output.Value := FALSE;
Assert.ThatBool(
	actual := output.Changed,
	message := "The reverse transition must also be pending"
).IsTrue();
output.ProcessOutput();
Assert.ThatBool(
	actual := output.Changed,
	message := "Processing acknowledges the reverse transition"
).IsFalse();
Assert.ThatBool(
	actual := rawOutput,
	message := "rawOutput should be FALSE"
).IsFalse();
END_METHOD

//! <summary>Borrows the concrete class name. Callers must not modify it.</summary>
{attribute 'monitoring' := 'call'}
PROPERTY ClassName : REFERENCE TO STRING
GET
ClassName REF= _ClassName;
END_GET
END_PROPERTY

//! <summary>Borrows the compiler-initialized namespace name. Callers must not modify it.</summary>
{attribute 'monitoring' := 'call'}
PROPERTY NamespaceName : REFERENCE TO STRING
GET
NamespaceName REF= CurrentNamespace.Name;
END_GET
END_PROPERTY

//! <summary>Reports the concrete instance size in bytes.</summary>
{attribute 'monitoring' := 'call'}
PROPERTY SelfSize : ULINT
GET
SelfSize := XSIZEOF(THIS^);
END_GET
END_PROPERTY

END_FUNCTION_BLOCK

// ---- Tests/Devices/IO/DigitalOutputNormallyClosedTest.TcPOU
(*
SPDX-FileCopyrightText: c 2026 Oleksandr Tiutyk <trofimich@gmail.com>
SPDX-License-Identifier: MIT
License: https://opensource.org/license/mit
*)

(*!
<summary>Checks normally closed output inversion in both directions.</summary>
<description>
Uses a live case-owned automation parent and fresh local device fixtures on every run.
The scenario reads and writes ordinary simulated storage within one task cycle.
</description>
*)

{attribute 'no_assign'}
{attribute 'no_explicit_call' := 'do not call this function block directly'}
FUNCTION_BLOCK DigitalOutputNormallyClosedTest EXTENDS TOF_Testing.SingleCycleTest
VAR_STAT
	{attribute 'hide'}
	_ClassName : STRING := __POUNAME();
END_VAR
VAR
	//! <summary>Live parent borrowed by the method-local simulated device.</summary>
	_AutomationRoot : MockAutomationController(name := "DevicesIORoot");
END_VAR

(*!
<summary>Checks normally closed output inversion in both directions.</summary>
*)
METHOD PROTECTED ExecuteTest
VAR
	output : TOF_Devices_IO.DigitalOutput(name := "DO_NC", parent := _AutomationRoot);
	rawOutput : BOOL;
END_VAR
output.Initialize();
output.ContactType := TOF_Devices_IO.CONTACT_TYPE.NORMALLY_CLOSED;
output.BindToIO(rawValue := rawOutput);

output.Value := TRUE;
output.ProcessOutput();
Assert.ThatBool(
	actual := rawOutput,
	message := "rawOutput should be inverted FALSE for NC contact"
).IsFalse();

output.Value := FALSE;
output.ProcessOutput();
Assert.ThatBool(
	actual := rawOutput,
	message := "rawOutput should be inverted TRUE for NC contact"
).IsTrue();
END_METHOD

//! <summary>Borrows the concrete class name. Callers must not modify it.</summary>
{attribute 'monitoring' := 'call'}
PROPERTY ClassName : REFERENCE TO STRING
GET
ClassName REF= _ClassName;
END_GET
END_PROPERTY

//! <summary>Borrows the compiler-initialized namespace name. Callers must not modify it.</summary>
{attribute 'monitoring' := 'call'}
PROPERTY NamespaceName : REFERENCE TO STRING
GET
NamespaceName REF= CurrentNamespace.Name;
END_GET
END_PROPERTY

//! <summary>Reports the concrete instance size in bytes.</summary>
{attribute 'monitoring' := 'call'}
PROPERTY SelfSize : ULINT
GET
SelfSize := XSIZEOF(THIS^);
END_GET
END_PROPERTY

END_FUNCTION_BLOCK

// ---- Tests/Devices/IO/DirectAnalogValueConverterTest.TcPOU
(*
SPDX-FileCopyrightText: c 2026 Oleksandr Tiutyk <trofimich@gmail.com>
SPDX-License-Identifier: MIT
License: https://opensource.org/license/mit
*)

(*!
<summary>Checks direct conversion of INT16, INT32 and REAL32 in both directions.</summary>
<description>
Uses fresh method-local fixtures in a single task cycle.
</description>
*)

{attribute 'no_assign'}
{attribute 'no_explicit_call' := 'do not call this function block directly'}
FUNCTION_BLOCK DirectAnalogValueConverterTest EXTENDS TOF_Testing.SingleCycleTest
VAR_STAT
	{attribute 'hide'}
	_ClassName : STRING := __POUNAME();
END_VAR

(*!
<summary>Checks direct conversion of INT16, INT32 and REAL32 in both directions.</summary>
*)
METHOD PROTECTED ExecuteTest
VAR
	converter : TOF_Devices_IO.DirectAnalogValueConverter;
	rawResult : TOF_Devices_IO.RAW_ANALOG_VALUE;
	engineeringValue : LREAL;
END_VAR
// INT16
rawResult := converter.ConvertAnalogValueToRawValue(
	analogValue := 1234.0,
	rawValueType := TOF_Devices_IO.RAW_ANALOG_VALUE_TYPE.INT16
);
Assert.ThatInt(
	actual := rawResult.Int16,
	message := "INT16 raw value 1:1"
).ToBe(expected := 1234);

engineeringValue := converter.ConvertRawValueToAnalogValue(
	rawValue := rawResult,
	rawValueType := TOF_Devices_IO.RAW_ANALOG_VALUE_TYPE.INT16
);
Assert.ThatLongReal(
	actual := engineeringValue,
	message := "INT16 analog value 1:1"
).ToBe(expected := 1234.0, tolerance := 0.001);

// INT32
rawResult := converter.ConvertAnalogValueToRawValue(
	analogValue := 100000.0,
	rawValueType := TOF_Devices_IO.RAW_ANALOG_VALUE_TYPE.INT32
);
Assert.ThatDInt(
	actual := rawResult.Int32,
	message := "INT32 raw value 1:1"
).ToBe(expected := 100000);

engineeringValue := converter.ConvertRawValueToAnalogValue(
	rawValue := rawResult,
	rawValueType := TOF_Devices_IO.RAW_ANALOG_VALUE_TYPE.INT32
);
Assert.ThatLongReal(
	actual := engineeringValue,
	message := "INT32 analog value 1:1"
).ToBe(expected := 100000.0, tolerance := 0.001);

// REAL32 preserves both sign and fraction.
rawResult := converter.ConvertAnalogValueToRawValue(
	analogValue := LREAL#-12.75,
	rawValueType := TOF_Devices_IO.RAW_ANALOG_VALUE_TYPE.REAL32
);

Assert.ThatReal(
	actual := rawResult.Real32,
	message := "Direct conversion must preserve the fractional REAL32 output"
).ToBe(expected := REAL#-12.75);

engineeringValue := converter.ConvertRawValueToAnalogValue(
	rawValue := rawResult,
	rawValueType := TOF_Devices_IO.RAW_ANALOG_VALUE_TYPE.REAL32
);

Assert.ThatLongReal(
	actual := engineeringValue,
	message := "Direct conversion must preserve the fractional REAL32 input"
).ToBe(expected := LREAL#-12.75);
END_METHOD

//! <summary>Borrows the concrete class name. Callers must not modify it.</summary>
{attribute 'monitoring' := 'call'}
PROPERTY ClassName : REFERENCE TO STRING
GET
ClassName REF= _ClassName;
END_GET
END_PROPERTY

//! <summary>Borrows the compiler-initialized namespace name. Callers must not modify it.</summary>
{attribute 'monitoring' := 'call'}
PROPERTY NamespaceName : REFERENCE TO STRING
GET
NamespaceName REF= CurrentNamespace.Name;
END_GET
END_PROPERTY

//! <summary>Reports the concrete instance size in bytes.</summary>
{attribute 'monitoring' := 'call'}
PROPERTY SelfSize : ULINT
GET
SelfSize := XSIZEOF(THIS^);
END_GET
END_PROPERTY

END_FUNCTION_BLOCK

// ---- Tests/Devices/IO/AnalogInputScalingAndScalarBindingTest.TcPOU
(*
SPDX-FileCopyrightText: c 2026 Oleksandr Tiutyk <trofimich@gmail.com>
SPDX-License-Identifier: MIT
License: https://opensource.org/license/mit
*)

(*!
<summary>Checks scalar INT16 binding and positive and negative input values.</summary>
<description>
Uses a live case-owned automation parent and fresh local device fixtures on every run.
The scenario reads and writes ordinary simulated storage within one task cycle.
</description>
*)

{attribute 'no_assign'}
{attribute 'no_explicit_call' := 'do not call this function block directly'}
FUNCTION_BLOCK AnalogInputScalingAndScalarBindingTest EXTENDS TOF_Testing.SingleCycleTest
VAR_STAT
	{attribute 'hide'}
	_ClassName : STRING := __POUNAME();
END_VAR
VAR
	//! <summary>Live parent borrowed by the method-local simulated device.</summary>
	_AutomationRoot : MockAutomationController(name := "DevicesIORoot");
END_VAR

(*!
<summary>Checks scalar INT16 binding and positive and negative input values.</summary>
*)
METHOD PROTECTED ExecuteTest
VAR
	converter : TOF_Devices_IO.DirectAnalogValueConverter;
	analogInput : TOF_Devices_IO.AnalogInput(name := "AI_Scalar", parent := _AutomationRoot, converter := converter);
	rawInput : INT;
END_VAR
analogInput.Initialize();
analogInput.BindToInt16Value(rawValue := rawInput);

Assert.ThatBool(
	actual := analogInput.BoundToIO,
	message := "AnalogInput should be BoundToIO after BindToInt16Value"
).IsTrue();

rawInput := 5678;
analogInput.ProcessInput();

Assert.ThatLongReal(
	actual := analogInput.Value,
	message := "AnalogInput.Value should match raw INT input"
).ToBe(expected := 5678.0, tolerance := 0.001);

Assert.ThatBool(
	actual := analogInput.HasError,
	message := "AnalogInput should work without error when status is unbound"
).IsFalse();

rawInput := INT#-1234;
analogInput.ProcessInput();

Assert.ThatLongReal(
	actual := analogInput.Value,
	message := "Scalar input processing must preserve the INT16 sign"
).ToBe(expected := LREAL#-1234.0);
END_METHOD

//! <summary>Borrows the concrete class name. Callers must not modify it.</summary>
{attribute 'monitoring' := 'call'}
PROPERTY ClassName : REFERENCE TO STRING
GET
ClassName REF= _ClassName;
END_GET
END_PROPERTY

//! <summary>Borrows the compiler-initialized namespace name. Callers must not modify it.</summary>
{attribute 'monitoring' := 'call'}
PROPERTY NamespaceName : REFERENCE TO STRING
GET
NamespaceName REF= CurrentNamespace.Name;
END_GET
END_PROPERTY

//! <summary>Reports the concrete instance size in bytes.</summary>
{attribute 'monitoring' := 'call'}
PROPERTY SelfSize : ULINT
GET
SelfSize := XSIZEOF(THIS^);
END_GET
END_PROPERTY

END_FUNCTION_BLOCK

// ---- Tests/Devices/IO/AnalogInputChannelStatusAndErrorReportingTest.TcPOU
(*
SPDX-FileCopyrightText: c 2026 Oleksandr Tiutyk <trofimich@gmail.com>
SPDX-License-Identifier: MIT
License: https://opensource.org/license/mit
*)

(*!
<summary>Checks channel diagnostics across processing, execution and rebinding.</summary>
<description>
Uses a live case-owned automation parent and fresh local device fixtures on every run.
The scenario reads and writes ordinary simulated storage within one task cycle.
</description>
*)

{attribute 'no_assign'}
{attribute 'no_explicit_call' := 'do not call this function block directly'}
FUNCTION_BLOCK AnalogInputChannelStatusAndErrorReportingTest EXTENDS TOF_Testing.SingleCycleTest
VAR CONSTANT
	//! <summary>Bit 6 is the simulated channel measurement or hardware error.</summary>
	_ChannelErrorStatus : WORD := WORD#16#0040;
	//! <summary>Expected diagnostic for a sampled channel error.</summary>
	_ChannelErrorMessage : WSTRING := "Analog input channel reports error";
END_VAR
VAR_STAT
	{attribute 'hide'}
	_ClassName : STRING := __POUNAME();
END_VAR
VAR
	//! <summary>Live parent borrowed by the method-local simulated device.</summary>
	_AutomationRoot : MockAutomationController(name := "DevicesIORoot");
END_VAR

(*!
<summary>Checks channel diagnostics across processing, execution and rebinding.</summary>
*)
METHOD PROTECTED ExecuteTest
VAR
	converter : TOF_Devices_IO.DirectAnalogValueConverter;
	analogInput : AnalogInputRecoveryProbe(name := "AI_Chan", parent := _AutomationRoot, converter := converter);
	//! <summary>Status word at offset 0 and signed 16-bit value bits at offset 1.</summary>
	channelData : ARRAY [0..1] OF WORD;
	channel : POINTER TO TOF_IOModels.ANALOG_INPUT_INT_CHANNEL;
	unboundChannel : REFERENCE TO TOF_IOModels.ANALOG_INPUT_INT_CHANNEL;
	i : INT;
END_VAR
Assert.ThatBool(
	actual := analogInput.Initialize(),
	message := "The analog input must initialize"
).IsTrue();

IF SIZEOF(channel^) <> SIZEOF(channelData) THEN
	RecordFailure(message := "The simulated INT16 channel must fit two words");

	RETURN;
END_IF

channel := ADR(channelData);
channelData[0] := WORD#16#0000;
channelData[1] := WORD#1000;
analogInput.BindToInt16IO(rawValues := channel^);
Assert.ThatBool(
	actual := analogInput.BoundToIO,
	message := "A valid simulated channel must bind"
).IsTrue();
Assert.ThatBool(
	actual := channelData[0] = WORD#16#0000 AND_THEN channelData[1] = WORD#1000,
	message := "Binding must leave both source words unchanged"
).IsTrue();
analogInput.ProcessInput();
analogInput.Execute();

Assert.ThatBool(
	actual := analogInput.HasError,
	message := "A healthy channel must have no error after the full cycle"
).IsFalse();

Assert.ThatLongReal(
	actual := analogInput.Value,
	message := "The bound component must read the simulated raw value"
).ToBe(expected := LREAL#1000.0);

// Hold bit 6 across two complete input and execution phases.
channelData[0] := _ChannelErrorStatus;

FOR i := 1 TO 2 DO
	analogInput.ProcessInput();

	Assert.ThatBool(
		actual := analogInput.Status.Error
				AND_THEN analogInput.StatusWord = _ChannelErrorStatus
				AND_THEN analogInput.HasError
				AND_THEN analogInput.Error.Severity = TOF_Core.ERROR_SEVERITY.ERROR
				AND_THEN analogInput.Error.TopMessage = _ChannelErrorMessage,
		message := "A sampled bit 6 must report the channel error after ProcessInput"
	).IsTrue();

	analogInput.Execute();

	Assert.ThatBool(
		actual := analogInput.StatusWord = _ChannelErrorStatus
				AND_THEN analogInput.HasError
				AND_THEN analogInput.Error.Severity = TOF_Core.ERROR_SEVERITY.ERROR
				AND_THEN analogInput.Error.TopMessage = _ChannelErrorMessage
				AND_THEN analogInput.OperationalState = TOF_Automation.OPERATIONAL_STATE.WORKING
				AND_THEN analogInput.RecoveryCalls = UDINT#0,
		message := "A persistent channel error must survive Execute without stopping or recovering the leaf"
	).IsTrue();
END_FOR

channelData[0] := WORD#0;
analogInput.ProcessInput();

Assert.ThatBool(
	actual := NOT analogInput.Status.Error AND_THEN analogInput.StatusWord = WORD#0 AND_THEN NOT analogInput.HasError,
	message := "Sampling a clear bit 6 must clear the channel diagnostic in the input phase"
).IsTrue();

analogInput.Execute();

Assert.ThatBool(
	actual := analogInput.StatusWord = WORD#0
		AND_THEN NOT analogInput.HasError
		AND_THEN analogInput.Error.Empty
		AND_THEN analogInput.RecoveryCalls = UDINT#0,
	message := "The recovered channel must remain clear after Execute without a recovery callback"
).IsTrue();

channelData[0] := _ChannelErrorStatus;
channelData[1] := WORD#2000;
analogInput.ProcessInput();
analogInput.Execute();
analogInput.BindToInt16IO(rawValues := unboundChannel);

Assert.ThatBool(
	actual := NOT analogInput.BoundToIO
		AND_THEN analogInput.StatusWord = _ChannelErrorStatus
		AND_THEN analogInput.HasError,
	message := "Unbinding clears the value link while keeping the last sample until input processing"
).IsTrue();

analogInput.ProcessInput();

Assert.ThatBool(
	actual := NOT analogInput.Status.Error AND_THEN analogInput.StatusWord = WORD#0 AND_THEN NOT analogInput.HasError,
	message := "Input processing without a status binding must clear the sampled status and channel error"
).IsTrue();

analogInput.Execute();

Assert.ThatBool(
	actual := analogInput.StatusWord = WORD#0
		AND_THEN NOT analogInput.HasError
		AND_THEN analogInput.Error.Empty
		AND_THEN analogInput.RecoveryCalls = UDINT#0,
	message := "The unbound input must remain clear after Execute"
).IsTrue();
Assert.ThatBool(
	actual := channelData[0] = WORD#16#0040 AND_THEN channelData[1] = WORD#2000,
	message := "Unbinding must leave source data unchanged"
).IsTrue();
channelData[0] := WORD#16#0000;
analogInput.BindToInt16IO(rawValues := channel^);
analogInput.ProcessInput();
Assert.ThatBool(
	actual := analogInput.BoundToIO,
	message := "A valid channel must bind again after unbinding"
).IsTrue();
Assert.ThatLongReal(
	actual := analogInput.Value,
	message := "Rebinding must read the current source value"
).ToBe(expected := LREAL#2000.0);
Assert.ThatBool(
	actual := channelData[0] = WORD#16#0000 AND_THEN channelData[1] = WORD#2000,
	message := "Input processing and rebinding must leave source data unchanged"
).IsTrue();
END_METHOD

//! <summary>Borrows the concrete class name. Callers must not modify it.</summary>
{attribute 'monitoring' := 'call'}
PROPERTY ClassName : REFERENCE TO STRING
GET
ClassName REF= _ClassName;
END_GET
END_PROPERTY

//! <summary>Borrows the compiler-initialized namespace name. Callers must not modify it.</summary>
{attribute 'monitoring' := 'call'}
PROPERTY NamespaceName : REFERENCE TO STRING
GET
NamespaceName REF= CurrentNamespace.Name;
END_GET
END_PROPERTY

//! <summary>Reports the concrete instance size in bytes.</summary>
{attribute 'monitoring' := 'call'}
PROPERTY SelfSize : ULINT
GET
SelfSize := XSIZEOF(THIS^);
END_GET
END_PROPERTY

END_FUNCTION_BLOCK

// ---- Tests/Devices/IO/AnalogInputRecoveryProbe.TcPOU
(*
SPDX-FileCopyrightText: © 2026 Oleksandr Tiutyk <trofimich@gmail.com>
SPDX-License-Identifier: MIT
License: https://opensource.org/license/mit
*)

(*!
<summary>Records automatic execution error recoveries for analog input tests.</summary>
<description>Uses the inherited analog input constructor, processing, and error handling.</description>
*)
{attribute 'no_explicit_call' := 'do not call this function block directly'}
FUNCTION_BLOCK FINAL AnalogInputRecoveryProbe EXTENDS TOF_Devices_IO.AnalogInput
VAR
	_RecoveryCalls : UDINT;
END_VAR

(*!
<summary>Counts the recovery callback issued by Execute().</summary>
*)
METHOD PROTECTED OnRecover
_RecoveryCalls := _RecoveryCalls + UDINT#1;
END_METHOD

(*!
<summary>Gets the number of recovery callbacks received by this instance.</summary>
*)
PROPERTY RecoveryCalls : UDINT
GET
RecoveryCalls := _RecoveryCalls;
END_GET
END_PROPERTY

END_FUNCTION_BLOCK

// ---- Tests/Devices/IO/AnalogInputConverterRecoveryTest.TcPOU
(*
SPDX-FileCopyrightText: c 2026 Oleksandr Tiutyk <trofimich@gmail.com>
SPDX-License-Identifier: MIT
License: https://opensource.org/license/mit
*)

(*!
<summary>Checks converter recovery and channel diagnostic precedence.</summary>
<description>
Uses a live case-owned automation parent and fresh local device fixtures on every run.
The scenario reads and writes ordinary simulated storage within one task cycle.
</description>
*)

{attribute 'no_assign'}
{attribute 'no_explicit_call' := 'do not call this function block directly'}
FUNCTION_BLOCK AnalogInputConverterRecoveryTest EXTENDS TOF_Testing.SingleCycleTest
VAR CONSTANT
	//! <summary>Bit 6 is the simulated channel measurement or hardware error.</summary>
	_ChannelErrorStatus : WORD := WORD#16#0040;
	//! <summary>Expected diagnostic for a sampled channel error.</summary>
	_ChannelErrorMessage : WSTRING := "Analog input channel reports error";
	//! <summary>Injected converter exception text used for diagnostic comparisons.</summary>
	_ConversionErrorMessage : WSTRING := "Injected analog input conversion failure.";
END_VAR
VAR_STAT
	{attribute 'hide'}
	_ClassName : STRING := __POUNAME();
END_VAR
VAR
	//! <summary>Live parent borrowed by the method-local simulated device.</summary>
	_AutomationRoot : MockAutomationController(name := "DevicesIORoot");
END_VAR

(*!
<summary>Checks converter recovery and channel diagnostic precedence.</summary>
*)
METHOD PROTECTED ExecuteTest
VAR
	converter : AnalogInputConverterProbe;
	analogInput : AnalogInputRecoveryProbe(
		name := "AI_ConversionRecovery",
		parent := _AutomationRoot,
		converter := converter
	);
	//! <summary>Simulated status word at offset 0 and signed INT value bits at offset 1.</summary>
	channelData : ARRAY [0..1] OF WORD;
	channel : POINTER TO TOF_IOModels.ANALOG_INPUT_INT_CHANNEL;
END_VAR
Assert.ThatBool(
	actual := analogInput.Initialize(),
	message := "The analog input must initialize"
).IsTrue();
analogInput.ExceptionHandlingPolicy := TOF_Core.ExceptionHandlingPolicies.SetErrorAndContinue;

IF SIZEOF(channel^) <> SIZEOF(channelData) THEN
	RecordFailure(message := "The simulated INT16 channel must fit two words");

	RETURN;
END_IF

channel := ADR(channelData);
channelData[0] := WORD#0;
channelData[1] := WORD#100;
analogInput.BindToInt16IO(rawValues := channel^);
analogInput.ProcessInput();
analogInput.Execute();
Assert.ThatBool(
	actual := analogInput.Value = LREAL#100.0,
	message := "The initial conversion must succeed"
).IsTrue();

converter.failureMessage := _ConversionErrorMessage;
channelData[1] := WORD#200;
analogInput.ProcessInput();
analogInput.Execute();

Assert.ThatBool(
	actual := analogInput.HasError
		AND_THEN analogInput.Error.Severity = TOF_Core.ERROR_SEVERITY.ERROR
		AND_THEN analogInput.Error.TopMessage = _ConversionErrorMessage,
	message := "Converter failure on a healthy channel must survive Execute"
).IsTrue();
Assert.ThatBool(
	actual := analogInput.Value = LREAL#100.0 AND_THEN analogInput.RecoveryCalls = UDINT#0,
	message := "A failed conversion must preserve the last value and defer recovery"
).IsTrue();

// Use different exception text to distinguish retaining the original error from copying a later one.
converter.failureMessage := "Repeated analog input conversion failure.";
channelData[0] := _ChannelErrorStatus;
analogInput.ProcessInput();
analogInput.Execute();

Assert.ThatBool(
	actual := analogInput.StatusWord = _ChannelErrorStatus
		AND_THEN analogInput.Error.TopMessage = _ConversionErrorMessage,
	message := "The converter diagnostic must take precedence while both errors are active"
).IsTrue();

channelData[0] := WORD#0;
analogInput.ProcessInput();
analogInput.Execute();

Assert.ThatBool(
	actual := analogInput.StatusWord = WORD#0
		AND_THEN analogInput.HasError
		AND_THEN analogInput.Error.Severity = TOF_Core.ERROR_SEVERITY.ERROR
		AND_THEN analogInput.Error.TopMessage = _ConversionErrorMessage
		AND_THEN analogInput.RecoveryCalls = UDINT#0,
	message := "Channel recovery must preserve the failing converter diagnostic"
).IsTrue();

converter.failureMessage := "";
analogInput.ProcessInput();

Assert.ThatBool(
	actual := analogInput.Value = LREAL#200.0
		AND_THEN analogInput.Error.TopMessage = _ConversionErrorMessage,
	message := "A successful input phase must update Value and leave recovery to Execute"
).IsTrue();

analogInput.Execute();

Assert.ThatBool(
	actual := NOT analogInput.HasError AND_THEN analogInput.RecoveryCalls = UDINT#1,
	message := "Execute must clear the recovered conversion error and call OnRecover once"
).IsTrue();

// A new conversion failure must be reported even when the channel fails in the same phase.
channelData[0] := _ChannelErrorStatus;
channelData[1] := WORD#300;
converter.failureMessage := _ConversionErrorMessage;
analogInput.ProcessInput();
analogInput.Execute();

Assert.ThatBool(
	actual := analogInput.StatusWord = _ChannelErrorStatus
		AND_THEN analogInput.Error.Severity = TOF_Core.ERROR_SEVERITY.ERROR
		AND_THEN analogInput.Error.TopMessage = _ConversionErrorMessage,
	message := "An active channel error must not block capture of a new conversion failure"
).IsTrue();

// Recover the converter first, with the channel fault still active.
converter.failureMessage := "";
analogInput.ProcessInput();
analogInput.Execute();

Assert.ThatBool(
	actual := analogInput.HasError
		AND_THEN analogInput.Error.TopMessage = _ChannelErrorMessage
		AND_THEN analogInput.Value = LREAL#300.0
		AND_THEN analogInput.RecoveryCalls = UDINT#2,
	message := "Converter recovery must expose the still-active channel error"
).IsTrue();

channelData[0] := WORD#0;
analogInput.ProcessInput();
analogInput.Execute();

Assert.ThatBool(
	actual := NOT analogInput.HasError AND_THEN analogInput.RecoveryCalls = UDINT#2,
	message := "Channel recovery must clear its diagnostic without another recovery callback"
).IsTrue();
END_METHOD

//! <summary>Borrows the concrete class name. Callers must not modify it.</summary>
{attribute 'monitoring' := 'call'}
PROPERTY ClassName : REFERENCE TO STRING
GET
ClassName REF= _ClassName;
END_GET
END_PROPERTY

//! <summary>Borrows the compiler-initialized namespace name. Callers must not modify it.</summary>
{attribute 'monitoring' := 'call'}
PROPERTY NamespaceName : REFERENCE TO STRING
GET
NamespaceName REF= CurrentNamespace.Name;
END_GET
END_PROPERTY

//! <summary>Reports the concrete instance size in bytes.</summary>
{attribute 'monitoring' := 'call'}
PROPERTY SelfSize : ULINT
GET
SelfSize := XSIZEOF(THIS^);
END_GET
END_PROPERTY

END_FUNCTION_BLOCK

// ---- Tests/Devices/IO/AnalogInputConverterProbe.TcPOU
(*
SPDX-FileCopyrightText: © 2026 Oleksandr Tiutyk <trofimich@gmail.com>
SPDX-License-Identifier: MIT
License: https://opensource.org/license/mit
*)

(*!
<summary>Provides pass-through conversion with a selectable input failure for diagnostics tests.</summary>
<description>Uses the direct converter for successful input conversion and all output conversion.</description>
*)
{attribute 'no_explicit_call' := 'do not call this function block directly'}
FUNCTION_BLOCK FINAL AnalogInputConverterProbe EXTENDS TOF_Devices_IO.DirectAnalogValueConverter
VAR_INPUT
	//! <summary>Raises a standard exception with this text on input conversion when the message is nonempty.</summary>
	failureMessage : TOF_Core.ERROR_MESSAGE;
END_VAR

(*!
<summary>Converts the raw input or raises the injected failure for the input's exception policy.</summary>
<param name="rawValue">Raw channel value.</param>
<param name="rawValueType">Representation of the raw value.</param>
*)
METHOD ConvertRawValueToAnalogValue : LREAL
VAR_INPUT
	rawValue : TOF_Devices_IO.RAW_ANALOG_VALUE;
	rawValueType : TOF_Devices_IO.RAW_ANALOG_VALUE_TYPE;
END_VAR
IF failureMessage <> "" THEN
	TOF_Core.Exceptions.ThrowStandard(
		sourceNamespaceName := NamespaceName,
		sourceClassName := ClassName,
		sourcePOUName := __POUNAME(),
		sourcePosition := __POSITION(),
		message := failureMessage
	);
END_IF

ConvertRawValueToAnalogValue := SUPER^.ConvertRawValueToAnalogValue(
	rawValue := rawValue,
	rawValueType := rawValueType
);
END_METHOD

END_FUNCTION_BLOCK

// ---- Tests/Devices/IO/AnalogInputCriticalConversionErrorTest.TcPOU
(*
SPDX-FileCopyrightText: c 2026 Oleksandr Tiutyk <trofimich@gmail.com>
SPDX-License-Identifier: MIT
License: https://opensource.org/license/mit
*)

(*!
<summary>Checks critical converter errors and explicit recovery through Reset.</summary>
<description>
Uses a live case-owned automation parent and fresh local device fixtures on every run.
The scenario reads and writes ordinary simulated storage within one task cycle.
</description>
*)

{attribute 'no_assign'}
{attribute 'no_explicit_call' := 'do not call this function block directly'}
FUNCTION_BLOCK AnalogInputCriticalConversionErrorTest EXTENDS TOF_Testing.SingleCycleTest
VAR CONSTANT
	//! <summary>Bit 6 is the simulated channel measurement or hardware error.</summary>
	_ChannelErrorStatus : WORD := WORD#16#0040;
	//! <summary>Injected converter exception text used for diagnostic comparisons.</summary>
	_ConversionErrorMessage : WSTRING := "Injected analog input conversion failure.";
END_VAR
VAR_STAT
	{attribute 'hide'}
	_ClassName : STRING := __POUNAME();
END_VAR
VAR
	//! <summary>Live parent borrowed by the method-local simulated device.</summary>
	_AutomationRoot : MockAutomationController(name := "DevicesIORoot");
END_VAR

(*!
<summary>Checks critical converter errors and explicit recovery through Reset.</summary>
*)
METHOD PROTECTED ExecuteTest
VAR
	converter : AnalogInputConverterProbe;
	analogInput : AnalogInputRecoveryProbe(
		name := "AI_CriticalConversion",
		parent := _AutomationRoot,
		converter := converter
	);
	//! <summary>Simulated status word at offset 0 and signed INT value bits at offset 1.</summary>
	channelData : ARRAY [0..1] OF WORD;
	channel : POINTER TO TOF_IOModels.ANALOG_INPUT_INT_CHANNEL;
END_VAR
Assert.ThatBool(
	actual := analogInput.Initialize(),
	message := "The analog input must initialize"
).IsTrue();
analogInput.ExceptionHandlingPolicy := TOF_Core.ExceptionHandlingPolicies.SetErrorAndStop;

IF SIZEOF(channel^) <> SIZEOF(channelData) THEN
	RecordFailure(message := "The simulated INT16 channel must fit two words");

	RETURN;
END_IF

channel := ADR(channelData);
channelData[0] := _ChannelErrorStatus;
channelData[1] := WORD#100;
analogInput.BindToInt16IO(rawValues := channel^);
converter.failureMessage := _ConversionErrorMessage;
analogInput.ProcessInput();
analogInput.Execute();

Assert.ThatBool(
	actual := analogInput.OperationalState = TOF_Automation.OPERATIONAL_STATE.STOPPED
		AND_THEN analogInput.HasError
		AND_THEN analogInput.Error.Severity = TOF_Core.ERROR_SEVERITY.CRITICAL
		AND_THEN analogInput.Error.TopMessage = _ConversionErrorMessage,
	message := "The critical conversion error must stop the leaf and take precedence over the channel error"
).IsTrue();

converter.failureMessage := "";
channelData[0] := WORD#0;
analogInput.ProcessInput();
analogInput.Execute();

Assert.ThatBool(
	actual := analogInput.OperationalState = TOF_Automation.OPERATIONAL_STATE.STOPPED
		AND_THEN analogInput.StatusWord = WORD#0
		AND_THEN analogInput.Value = LREAL#100.0
		AND_THEN analogInput.HasError
		AND_THEN analogInput.Error.Severity = TOF_Core.ERROR_SEVERITY.CRITICAL
		AND_THEN analogInput.Error.TopMessage = _ConversionErrorMessage,
	message := "Successful input with a healthy channel must preserve the critical diagnostic while stopped"
).IsTrue();

analogInput.Reset();
analogInput.Execute();

Assert.ThatBool(
	actual := analogInput.OperationalState = TOF_Automation.OPERATIONAL_STATE.WORKING
		AND_THEN NOT analogInput.HasError
		AND_THEN analogInput.RecoveryCalls = UDINT#0,
	message := "Reset must clear the critical diagnostic and restore WORKING"
).IsTrue();
END_METHOD

//! <summary>Borrows the concrete class name. Callers must not modify it.</summary>
{attribute 'monitoring' := 'call'}
PROPERTY ClassName : REFERENCE TO STRING
GET
ClassName REF= _ClassName;
END_GET
END_PROPERTY

//! <summary>Borrows the compiler-initialized namespace name. Callers must not modify it.</summary>
{attribute 'monitoring' := 'call'}
PROPERTY NamespaceName : REFERENCE TO STRING
GET
NamespaceName REF= CurrentNamespace.Name;
END_GET
END_PROPERTY

//! <summary>Reports the concrete instance size in bytes.</summary>
{attribute 'monitoring' := 'call'}
PROPERTY SelfSize : ULINT
GET
SelfSize := XSIZEOF(THIS^);
END_GET
END_PROPERTY

END_FUNCTION_BLOCK

// ---- Tests/Devices/IO/AnalogInputStatusWordIsolationTest.TcPOU
(*
SPDX-FileCopyrightText: c 2026 Oleksandr Tiutyk <trofimich@gmail.com>
SPDX-License-Identifier: MIT
License: https://opensource.org/license/mit
*)

(*!
<summary>Checks sampled status isolation through the read-only input interface.</summary>
<description>
Uses a live case-owned automation parent and fresh local device fixtures on every run.
The scenario reads and writes ordinary simulated storage within one task cycle.
</description>
*)

{attribute 'no_assign'}
{attribute 'no_explicit_call' := 'do not call this function block directly'}
FUNCTION_BLOCK AnalogInputStatusWordIsolationTest EXTENDS TOF_Testing.SingleCycleTest
VAR CONSTANT
	//! <summary>Bit 6 is the simulated channel measurement or hardware error.</summary>
	_ChannelErrorStatus : WORD := WORD#16#0040;
	//! <summary>Expected diagnostic for a sampled channel error.</summary>
	_ChannelErrorMessage : WSTRING := "Analog input channel reports error";
END_VAR
VAR_STAT
	{attribute 'hide'}
	_ClassName : STRING := __POUNAME();
END_VAR
VAR
	//! <summary>Live parent borrowed by the method-local simulated device.</summary>
	_AutomationRoot : MockAutomationController(name := "DevicesIORoot");
END_VAR

(*!
<summary>Checks sampled status isolation through the read-only input interface.</summary>
*)
METHOD PROTECTED ExecuteTest
VAR
	converter : TOF_Devices_IO.DirectAnalogValueConverter;
	analogInput : TOF_Devices_IO.AnalogInput(name := "AI_StatusWord", parent := _AutomationRoot, converter := converter);
	inputView : TOF_Devices_IO.IReadOnlyAnalogInput;
	statusProvider : TOF_Devices_IO.IAnalogInputStatusProvider;
	legacyStatus : REFERENCE TO TOF_Devices_IO.ANALOG_INPUT_STATUS;
	statusCopy : WORD;
	//! <summary>Simulated status word at offset 0 and signed INT value bits at offset 1.</summary>
	channelData : ARRAY [0..1] OF WORD;
	channel : POINTER TO TOF_IOModels.ANALOG_INPUT_INT_CHANNEL;
END_VAR
Assert.ThatBool(
	actual := analogInput.Initialize(),
	message := "The analog input must initialize"
).IsTrue();
inputView := analogInput;

IF NOT __QUERYINTERFACE(inputView, statusProvider) OR_ELSE statusProvider = 0 THEN
	Assert.ThatBool(
		actual := FALSE,
		message := "IReadOnlyAnalogInput must support querying IAnalogInputStatusProvider"
	).IsTrue();

	RETURN;
END_IF

Assert.ThatBool(
	actual := statusProvider.StatusWord = WORD#0,
	message := "StatusWord must start at zero"
).IsTrue();

IF SIZEOF(channel^) <> SIZEOF(channelData) THEN
	RecordFailure(message := "The simulated INT16 channel must fit two words");

	RETURN;
END_IF

channel := ADR(channelData);
channelData[0] := _ChannelErrorStatus;
channelData[1] := WORD#0;
analogInput.BindToInt16IO(rawValues := channel^);
inputView.ProcessInput();

legacyStatus REF= inputView.Status;

IF NOT __ISVALIDREF(legacyStatus) THEN
	RecordFailure(message := "The legacy status reference must be valid");

	RETURN;
END_IF

legacyStatus.SetStatus(status := WORD#0);
statusCopy := statusProvider.StatusWord;
statusCopy.6 := FALSE;
inputView.Execute();

Assert.ThatBool(
	actual := statusCopy = WORD#0
		AND_THEN NOT inputView.Status.Error
		AND_THEN statusProvider.StatusWord = _ChannelErrorStatus
		AND_THEN inputView.HasError
		AND_THEN inputView.Error.TopMessage = _ChannelErrorMessage,
	message := "Mutating the legacy view or local copy must leave the sampled word and diagnostic intact"
).IsTrue();

inputView.ProcessInput();
inputView.Execute();

Assert.ThatBool(
	actual := inputView.Status.Error AND_THEN statusProvider.StatusWord = _ChannelErrorStatus,
	message := "Input processing must refresh the legacy view from the sampled word"
).IsTrue();
END_METHOD

//! <summary>Borrows the concrete class name. Callers must not modify it.</summary>
{attribute 'monitoring' := 'call'}
PROPERTY ClassName : REFERENCE TO STRING
GET
ClassName REF= _ClassName;
END_GET
END_PROPERTY

//! <summary>Borrows the compiler-initialized namespace name. Callers must not modify it.</summary>
{attribute 'monitoring' := 'call'}
PROPERTY NamespaceName : REFERENCE TO STRING
GET
NamespaceName REF= CurrentNamespace.Name;
END_GET
END_PROPERTY

//! <summary>Reports the concrete instance size in bytes.</summary>
{attribute 'monitoring' := 'call'}
PROPERTY SelfSize : ULINT
GET
SelfSize := XSIZEOF(THIS^);
END_GET
END_PROPERTY

END_FUNCTION_BLOCK

// ---- Tests/Devices/IO/AnalogInputStatusBitDecodingTest.TcPOU
(*
SPDX-FileCopyrightText: c 2026 Oleksandr Tiutyk <trofimich@gmail.com>
SPDX-License-Identifier: MIT
License: https://opensource.org/license/mit
*)

(*!
<summary>Checks status flags for individual bits and their reset.</summary>
<description>
Uses fresh method-local fixtures in a single task cycle.
</description>
*)

{attribute 'no_assign'}
{attribute 'no_explicit_call' := 'do not call this function block directly'}
FUNCTION_BLOCK AnalogInputStatusBitDecodingTest EXTENDS TOF_Testing.SingleCycleTest
VAR_STAT
	{attribute 'hide'}
	_ClassName : STRING := __POUNAME();
END_VAR

(*!
<summary>Checks status flags for individual bits and their reset.</summary>
*)
METHOD PROTECTED ExecuteTest
VAR
	status : TOF_Devices_IO.ANALOG_INPUT_STATUS;
END_VAR
status.SetStatus(status := 16#0001);
Assert.ThatBool(
	actual := status.Underrange,
	message := "Bit 0 must be Underrange"
).IsTrue();

status.SetStatus(status := 16#0002);
Assert.ThatBool(
	actual := status.Overrange,
	message := "Bit 1 must be Overrange"
).IsTrue();

status.SetStatus(status := 16#0004);
Assert.ThatBool(
	actual := status.ValueSmallerOrEqualLimit1,
	message := "Bit 2 must be Limit 1 smaller"
).IsTrue();

status.SetStatus(status := 16#0008);
Assert.ThatBool(
	actual := status.ValueBiggerOrEqualLimit1,
	message := "Bit 3 must be Limit 1 bigger"
).IsTrue();

status.SetStatus(status := 16#0010);
Assert.ThatBool(
	actual := status.ValueSmallerOrEqualLimit2,
	message := "Bit 4 must be Limit 2 smaller"
).IsTrue();

status.SetStatus(status := 16#0020);
Assert.ThatBool(
	actual := status.ValueBiggerOrEqualLimit2,
	message := "Bit 5 must be Limit 2 bigger"
).IsTrue();

status.SetStatus(status := 16#0040);
Assert.ThatBool(
	actual := status.Error,
	message := "Bit 6 must be Error"
).IsTrue();
Assert.ThatBool(
	actual := status.TxPDOState,
	message := "Bit 6 must NOT be TxPDOState"
).IsFalse();

status.SetStatus(status := 16#4000);
Assert.ThatBool(
	actual := status.TxPDOState,
	message := "Bit 14 must be TxPDOState"
).IsTrue();
Assert.ThatBool(
	actual := status.Error,
	message := "Bit 14 must NOT be Error"
).IsFalse();

status.SetStatus(status := 16#8000);
Assert.ThatBool(
	actual := status.TxPDOToggle,
	message := "Bit 15 must be TxPDOToggle"
).IsTrue();

status.SetStatus(status := WORD#16#C040);

Assert.ThatBool(
	actual := status.Error AND_THEN status.TxPDOState AND_THEN status.TxPDOToggle,
	message := "Bits 6, 14 and 15 must be independently active together"
).IsTrue();

status.SetStatus(status := WORD#0);

Assert.ThatBool(
	actual := NOT status.Error AND_THEN NOT status.TxPDOState AND_THEN NOT status.TxPDOToggle,
	message := "A zero status word must clear all three diagnostic flags"
).IsTrue();
END_METHOD

//! <summary>Borrows the concrete class name. Callers must not modify it.</summary>
{attribute 'monitoring' := 'call'}
PROPERTY ClassName : REFERENCE TO STRING
GET
ClassName REF= _ClassName;
END_GET
END_PROPERTY

//! <summary>Borrows the compiler-initialized namespace name. Callers must not modify it.</summary>
{attribute 'monitoring' := 'call'}
PROPERTY NamespaceName : REFERENCE TO STRING
GET
NamespaceName REF= CurrentNamespace.Name;
END_GET
END_PROPERTY

//! <summary>Reports the concrete instance size in bytes.</summary>
{attribute 'monitoring' := 'call'}
PROPERTY SelfSize : ULINT
GET
SelfSize := XSIZEOF(THIS^);
END_GET
END_PROPERTY

END_FUNCTION_BLOCK

// ---- Tests/Devices/IO/AnalogOutputScalingTest.TcPOU
(*
SPDX-FileCopyrightText: c 2026 Oleksandr Tiutyk <trofimich@gmail.com>
SPDX-License-Identifier: MIT
License: https://opensource.org/license/mit
*)

(*!
<summary>Checks direct analog output processing for a bound INT16 value.</summary>
<description>
Uses a live case-owned automation parent and fresh local device fixtures on every run.
The scenario reads and writes ordinary simulated storage within one task cycle.
</description>
*)

{attribute 'no_assign'}
{attribute 'no_explicit_call' := 'do not call this function block directly'}
FUNCTION_BLOCK AnalogOutputScalingTest EXTENDS TOF_Testing.SingleCycleTest
VAR_STAT
	{attribute 'hide'}
	_ClassName : STRING := __POUNAME();
END_VAR
VAR
	//! <summary>Live parent borrowed by the method-local simulated device.</summary>
	_AutomationRoot : MockAutomationController(name := "DevicesIORoot");
END_VAR

(*!
<summary>Checks direct analog output processing for a bound INT16 value.</summary>
*)
METHOD PROTECTED ExecuteTest
VAR
	converter : TOF_Devices_IO.DirectAnalogValueConverter;
	analogOutput : TOF_Devices_IO.AnalogOutput(name := "AO_Test", parent := _AutomationRoot, converter := converter);
	rawOutput : INT;
END_VAR
analogOutput.Initialize();
analogOutput.BindToInt16IO(rawVariable := rawOutput);

analogOutput.Value := 750.0;
analogOutput.ProcessOutput();

Assert.ThatInt(
	actual := rawOutput,
	message := "Raw INT output should match 750"
).ToBe(expected := 750);
END_METHOD

//! <summary>Borrows the concrete class name. Callers must not modify it.</summary>
{attribute 'monitoring' := 'call'}
PROPERTY ClassName : REFERENCE TO STRING
GET
ClassName REF= _ClassName;
END_GET
END_PROPERTY

//! <summary>Borrows the compiler-initialized namespace name. Callers must not modify it.</summary>
{attribute 'monitoring' := 'call'}
PROPERTY NamespaceName : REFERENCE TO STRING
GET
NamespaceName REF= CurrentNamespace.Name;
END_GET
END_PROPERTY

//! <summary>Reports the concrete instance size in bytes.</summary>
{attribute 'monitoring' := 'call'}
PROPERTY SelfSize : ULINT
GET
SelfSize := XSIZEOF(THIS^);
END_GET
END_PROPERTY

END_FUNCTION_BLOCK

// ---- Tests/Devices/IO/AnalogOutputEqualRawLimitsTest.TcPOU
(*
SPDX-FileCopyrightText: c 2026 Oleksandr Tiutyk <trofimich@gmail.com>
SPDX-License-Identifier: MIT
License: https://opensource.org/license/mit
*)

(*!
<summary>Checks output with equal raw limits for INT16, INT32 and REAL32.</summary>
<description>
Uses a live case-owned automation parent and fresh local device fixtures on every run.
The scenario reads and writes ordinary simulated storage within one task cycle.
</description>
*)

{attribute 'no_assign'}
{attribute 'no_explicit_call' := 'do not call this function block directly'}
FUNCTION_BLOCK AnalogOutputEqualRawLimitsTest EXTENDS TOF_Testing.SingleCycleTest
VAR_STAT
	{attribute 'hide'}
	_ClassName : STRING := __POUNAME();
END_VAR
VAR
	//! <summary>Live parent borrowed by the method-local simulated device.</summary>
	_AutomationRoot : MockAutomationController(name := "DevicesIORoot");
END_VAR

(*!
<summary>Checks output with equal raw limits for INT16, INT32 and REAL32.</summary>
*)
METHOD PROTECTED ExecuteTest
VAR
	minEngineeringValue : LREAL := 0.0;
	maxEngineeringValue : LREAL := 100.0;
	minRawValue : TOF_Devices_IO.RAW_ANALOG_VALUE;
	maxRawValue : TOF_Devices_IO.RAW_ANALOG_VALUE;
	converter : TOF_Devices_IO.DynamicRangeAnalogValueConverter(
		minAnalogValue := minEngineeringValue,
		maxAnalogValue := maxEngineeringValue,
		minRawValue := minRawValue,
		maxRawValue := maxRawValue
	);
	analogOutput : TOF_Devices_IO.AnalogOutput(
		name := "AO_EqualRawLimits",
		parent := _AutomationRoot,
		converter := converter
	);

	rawInt16Output : INT;
	rawInt32Output : DINT;
	rawReal32Output : REAL;
	convertedValue : TOF_Devices_IO.RAW_ANALOG_VALUE;
END_VAR
analogOutput.Initialize();
analogOutput.Value := 50.0;

// Fill the upper two bytes of the INT16 limit to verify that they are cleared in the result.
minRawValue.Int32 := DINT#16#12340000;
minRawValue.Int16 := INT#-1;
maxRawValue := minRawValue;

analogOutput.BindToInt16IO(rawVariable := rawInt16Output);
analogOutput.ProcessOutput();

Assert.ThatInt(
	actual := rawInt16Output,
	message := "Equal INT16 limits must be written to the bound INT output"
).ToBe(expected := INT#-1);

convertedValue := converter.ConvertAnalogValueToRawValue(
	analogValue := analogOutput.Value,
	rawValueType := TOF_Devices_IO.RAW_ANALOG_VALUE_TYPE.INT16
);

Assert.ThatDInt(
	actual := convertedValue.Int32,
	message := "The INT16 result must have zero upper bytes"
).ToBe(expected := DINT#16#0000FFFF);

minRawValue.Int32 := DINT#-1;
maxRawValue := minRawValue;

analogOutput.BindToInt32IO(rawVariable := rawInt32Output);
analogOutput.ProcessOutput();

Assert.ThatDInt(
	actual := rawInt32Output,
	message := "Equal INT32 limits must be written to the bound DINT output"
).ToBe(expected := DINT#-1);

minRawValue.Real32 := REAL#1.0;
maxRawValue := minRawValue;

analogOutput.BindToReal32IO(rawVariable := rawReal32Output);
analogOutput.ProcessOutput();

Assert.ThatReal(
	actual := rawReal32Output,
	message := "Equal REAL32 limits must be written to the bound REAL output"
).ToBe(expected := REAL#1.0);
END_METHOD

//! <summary>Borrows the concrete class name. Callers must not modify it.</summary>
{attribute 'monitoring' := 'call'}
PROPERTY ClassName : REFERENCE TO STRING
GET
ClassName REF= _ClassName;
END_GET
END_PROPERTY

//! <summary>Borrows the compiler-initialized namespace name. Callers must not modify it.</summary>
{attribute 'monitoring' := 'call'}
PROPERTY NamespaceName : REFERENCE TO STRING
GET
NamespaceName REF= CurrentNamespace.Name;
END_GET
END_PROPERTY

//! <summary>Reports the concrete instance size in bytes.</summary>
{attribute 'monitoring' := 'call'}
PROPERTY SelfSize : ULINT
GET
SelfSize := XSIZEOF(THIS^);
END_GET
END_PROPERTY

END_FUNCTION_BLOCK

// ---- Tests/Devices/IO/DynamicRangeAnalogValueConverterTest.TcPOU
(*
SPDX-FileCopyrightText: c 2026 Oleksandr Tiutyk <trofimich@gmail.com>
SPDX-License-Identifier: MIT
License: https://opensource.org/license/mit
*)

(*!
<summary>Checks live changes of referenced engineering and raw limits.</summary>
<description>
Uses fresh method-local fixtures in a single task cycle.
</description>
*)

{attribute 'no_assign'}
{attribute 'no_explicit_call' := 'do not call this function block directly'}
FUNCTION_BLOCK DynamicRangeAnalogValueConverterTest EXTENDS TOF_Testing.SingleCycleTest
VAR_STAT
	{attribute 'hide'}
	_ClassName : STRING := __POUNAME();
END_VAR

(*!
<summary>Checks live changes of referenced engineering and raw limits.</summary>
*)
METHOD PROTECTED ExecuteTest
VAR
	minimumEngineeringValue : LREAL := 0.0;
	maximumEngineeringValue : LREAL := 100.0;
	minimumRawValue : TOF_Devices_IO.RAW_ANALOG_VALUE;
	maximumRawValue : TOF_Devices_IO.RAW_ANALOG_VALUE;
	converter : TOF_Devices_IO.DynamicRangeAnalogValueConverter(
		minAnalogValue := minimumEngineeringValue,
		maxAnalogValue := maximumEngineeringValue,
		minRawValue := minimumRawValue,
		maxRawValue := maximumRawValue
	);
	rawResult : TOF_Devices_IO.RAW_ANALOG_VALUE;
END_VAR
minimumRawValue.Int32 := 0;
minimumRawValue.Int16 := 0;
maximumRawValue.Int32 := 0;
maximumRawValue.Int16 := 1000;

rawResult := converter.ConvertAnalogValueToRawValue(
	analogValue := 50.0,
	rawValueType := TOF_Devices_IO.RAW_ANALOG_VALUE_TYPE.INT16
);
Assert.ThatInt(
	actual := rawResult.Int16,
	message := "Initial dynamic scale"
).ToBe(expected := 500);

// Change the referenced engineering limit.
maximumEngineeringValue := 200.0;

rawResult := converter.ConvertAnalogValueToRawValue(
	analogValue := 50.0,
	rawValueType := TOF_Devices_IO.RAW_ANALOG_VALUE_TYPE.INT16
);
Assert.ThatInt(
	actual := rawResult.Int16,
	message := "Dynamically updated scale"
).ToBe(expected := 250);

maximumRawValue.Int16 := INT#2000;
rawResult := converter.ConvertAnalogValueToRawValue(
	analogValue := LREAL#50.0,
	rawValueType := TOF_Devices_IO.RAW_ANALOG_VALUE_TYPE.INT16
);

Assert.ThatInt(
	actual := rawResult.Int16,
	message := "Changing the referenced raw maximum must update the scale"
).ToBe(expected := INT#500);
END_METHOD

//! <summary>Borrows the concrete class name. Callers must not modify it.</summary>
{attribute 'monitoring' := 'call'}
PROPERTY ClassName : REFERENCE TO STRING
GET
ClassName REF= _ClassName;
END_GET
END_PROPERTY

//! <summary>Borrows the compiler-initialized namespace name. Callers must not modify it.</summary>
{attribute 'monitoring' := 'call'}
PROPERTY NamespaceName : REFERENCE TO STRING
GET
NamespaceName REF= CurrentNamespace.Name;
END_GET
END_PROPERTY

//! <summary>Reports the concrete instance size in bytes.</summary>
{attribute 'monitoring' := 'call'}
PROPERTY SelfSize : ULINT
GET
SelfSize := XSIZEOF(THIS^);
END_GET
END_PROPERTY

END_FUNCTION_BLOCK

// ---- Tests/Devices/IO/StaticConverterCopiesLimitsTest.TcPOU
(*
SPDX-FileCopyrightText: c 2026 Oleksandr Tiutyk <trofimich@gmail.com>
SPDX-License-Identifier: MIT
License: https://opensource.org/license/mit
*)

(*!
<summary>Checks independent copies of the configured converter limits.</summary>
<description>
Uses fresh method-local fixtures in a single task cycle.
</description>
*)

{attribute 'no_assign'}
{attribute 'no_explicit_call' := 'do not call this function block directly'}
FUNCTION_BLOCK StaticConverterCopiesLimitsTest EXTENDS TOF_Testing.SingleCycleTest
VAR_STAT
	{attribute 'hide'}
	_ClassName : STRING := __POUNAME();
END_VAR

(*!
<summary>Checks independent copies of the configured converter limits.</summary>
*)
METHOD PROTECTED ExecuteTest
VAR
	minRaw : TOF_Devices_IO.RAW_ANALOG_VALUE;
	maxRaw : TOF_Devices_IO.RAW_ANALOG_VALUE := TOF_Devices_IO.RawAnalogValues.FromInt16(value := 1000);
	converter : TOF_Devices_IO.StaticRangeAnalogValueConverter(
		minAnalogValue := 0.0,
		maxAnalogValue := 100.0,
		minRawValue := minRaw,
		maxRawValue := maxRaw
	);
	resultRaw : TOF_Devices_IO.RAW_ANALOG_VALUE;
END_VAR
// Changing source unions must not change the stored constructor limits.
maxRaw.Int32 := 0;

Assert.ThatLongReal(
	actual := converter.MaxAnalogValue,
	message := "Constructor must preserve the configured analog maximum"
).ToBe(expected := 100.0, tolerance := 0.001);

resultRaw := converter.ConvertAnalogValueToRawValue(
	analogValue := 50.0,
	rawValueType := TOF_Devices_IO.RAW_ANALOG_VALUE_TYPE.INT16
);

Assert.ThatInt(
	actual := resultRaw.Int16,
	message := "Conversion must use copied raw limits after the source changes"
).ToBe(expected := 500);
END_METHOD

//! <summary>Borrows the concrete class name. Callers must not modify it.</summary>
{attribute 'monitoring' := 'call'}
PROPERTY ClassName : REFERENCE TO STRING
GET
ClassName REF= _ClassName;
END_GET
END_PROPERTY

//! <summary>Borrows the compiler-initialized namespace name. Callers must not modify it.</summary>
{attribute 'monitoring' := 'call'}
PROPERTY NamespaceName : REFERENCE TO STRING
GET
NamespaceName REF= CurrentNamespace.Name;
END_GET
END_PROPERTY

//! <summary>Reports the concrete instance size in bytes.</summary>
{attribute 'monitoring' := 'call'}
PROPERTY SelfSize : ULINT
GET
SelfSize := XSIZEOF(THIS^);
END_GET
END_PROPERTY

END_FUNCTION_BLOCK

// ---- Tests/Devices/IO/RangeConverterBoundaryClampingAndZeroDivisionTest.TcPOU
(*
SPDX-FileCopyrightText: c 2026 Oleksandr Tiutyk <trofimich@gmail.com>
SPDX-License-Identifier: MIT
License: https://opensource.org/license/mit
*)

(*!
<summary>Checks clamping and conversion with equal limits.</summary>
<description>
Uses fresh method-local fixtures in a single task cycle.
</description>
*)

{attribute 'no_assign'}
{attribute 'no_explicit_call' := 'do not call this function block directly'}
FUNCTION_BLOCK RangeConverterBoundaryClampingAndZeroDivisionTest EXTENDS TOF_Testing.SingleCycleTest
VAR_STAT
	{attribute 'hide'}
	_ClassName : STRING := __POUNAME();
END_VAR

(*!
<summary>Checks clamping and conversion with equal limits.</summary>
*)
METHOD PROTECTED ExecuteTest
VAR
	minRaw : TOF_Devices_IO.RAW_ANALOG_VALUE;
	clampingConverter : TOF_Devices_IO.StaticRangeAnalogValueConverter(
		minAnalogValue := 0.0,
		maxAnalogValue := 100.0,
		minRawValue := TOF_Devices_IO.RawAnalogValues.FromInt16(value := 0),
		maxRawValue := TOF_Devices_IO.RawAnalogValues.FromInt16(value := 1000)
	);
	equalLimitsConverter : TOF_Devices_IO.StaticRangeAnalogValueConverter(
		minAnalogValue := 0.0,
		maxAnalogValue := 0.0,
		minRawValue := TOF_Devices_IO.RawAnalogValues.FromInt16(value := 0),
		maxRawValue := TOF_Devices_IO.RawAnalogValues.FromInt16(value := 0)
	);
	rawResult : TOF_Devices_IO.RAW_ANALOG_VALUE;
	analogResult : LREAL;
END_VAR
minRaw.Int32 := 0;
minRaw.Int16 := 0;

// Test clamping above maximum
rawResult := clampingConverter.ConvertAnalogValueToRawValue(
	analogValue := 150.0,
	rawValueType := TOF_Devices_IO.RAW_ANALOG_VALUE_TYPE.INT16
);
Assert.ThatInt(
	actual := rawResult.Int16,
	message := "Clamped to max limit"
).ToBe(expected := 1000);

// Test clamping below minimum
rawResult := clampingConverter.ConvertAnalogValueToRawValue(
	analogValue := -50.0,
	rawValueType := TOF_Devices_IO.RAW_ANALOG_VALUE_TYPE.INT16
);
Assert.ThatInt(
	actual := rawResult.Int16,
	message := "Clamped to min limit"
).ToBe(expected := 0);

// Test equal limits (0 to 0) defense against Division by Zero
analogResult := equalLimitsConverter.ConvertRawValueToAnalogValue(
	rawValue := minRaw,
	rawValueType := TOF_Devices_IO.RAW_ANALOG_VALUE_TYPE.INT16
);
Assert.ThatLongReal(
	actual := analogResult,
	message := "Equal limits must safely return without Division by Zero"
).ToBe(expected := 0.0, tolerance := 0.001);
END_METHOD

//! <summary>Borrows the concrete class name. Callers must not modify it.</summary>
{attribute 'monitoring' := 'call'}
PROPERTY ClassName : REFERENCE TO STRING
GET
ClassName REF= _ClassName;
END_GET
END_PROPERTY

//! <summary>Borrows the compiler-initialized namespace name. Callers must not modify it.</summary>
{attribute 'monitoring' := 'call'}
PROPERTY NamespaceName : REFERENCE TO STRING
GET
NamespaceName REF= CurrentNamespace.Name;
END_GET
END_PROPERTY

//! <summary>Reports the concrete instance size in bytes.</summary>
{attribute 'monitoring' := 'call'}
PROPERTY SelfSize : ULINT
GET
SelfSize := XSIZEOF(THIS^);
END_GET
END_PROPERTY

END_FUNCTION_BLOCK

// ---- Tests/Collections/Contract/CollectionsContractTestGroup.TcPOU
(*
SPDX-FileCopyrightText: c 2026 Oleksandr Tiutyk <trofimich@gmail.com>
SPDX-License-Identifier: MIT
License: https://opensource.org/license/mit
*)

(*!
<summary>Runs the collection contract cases in their original scenario order.</summary>
<description>
Owns the shared fixture, its child cases and fixed registration array. The cases run sequentially.
Keep the group at a stable address in its owner task.
</description>
*)

{attribute 'no_assign'}
{attribute 'no_explicit_call' := 'do not call this function block directly'}
FUNCTION_BLOCK CollectionsContractTestGroup EXTENDS TOF_Testing.TestGroup<22>
VAR_STAT
	{attribute 'hide'}
	_ClassName : STRING := __POUNAME();
END_VAR
VAR
	_Fixture : CollectionsContractTestFixture;

	_CopyFailurePreservesException : CollectionsContractTestCase(
		name := "CopyFailurePreservesException",
		parent := THIS^,
		fixture := _Fixture,
		scenario := COLLECTIONS_CONTRACT_SCENARIO.COPY_FAILURE_PRESERVES_EXCEPTION
	);
	_SecondCopyFailureCleanup : CollectionsContractTestCase(
		name := "SecondCopyFailureCleanup",
		parent := THIS^,
		fixture := _Fixture,
		scenario := COLLECTIONS_CONTRACT_SCENARIO.SECOND_COPY_FAILURE_CLEANUP
	);
	_StaticFullCopyCleanup : CollectionsContractTestCase(
		name := "StaticFullCopyCleanup",
		parent := THIS^,
		fixture := _Fixture,
		scenario := COLLECTIONS_CONTRACT_SCENARIO.STATIC_FULL_COPY_CLEANUP
	);
	_ByteOverlapAndBounds : CollectionsContractTestCase(
		name := "ByteOverlapAndBounds",
		parent := THIS^,
		fixture := _Fixture,
		scenario := COLLECTIONS_CONTRACT_SCENARIO.BYTE_OVERLAP_AND_BOUNDS
	);
	_ByteSizeRejections : CollectionsContractTestCase(
		name := "ByteSizeRejections",
		parent := THIS^,
		fixture := _Fixture,
		scenario := COLLECTIONS_CONTRACT_SCENARIO.BYTE_SIZE_REJECTIONS
	);
	_ListOwnershipReplacement : CollectionsContractTestCase(
		name := "ListOwnershipReplacement",
		parent := THIS^,
		fixture := _Fixture,
		scenario := COLLECTIONS_CONTRACT_SCENARIO.LIST_OWNERSHIP_REPLACEMENT
	);
	_ListRemovalLimits : CollectionsContractTestCase(
		name := "ListRemovalLimits",
		parent := THIS^,
		fixture := _Fixture,
		scenario := COLLECTIONS_CONTRACT_SCENARIO.LIST_REMOVAL_LIMITS
	);
	_SortFailurePreservesEntries : CollectionsContractTestCase(
		name := "SortFailurePreservesEntries",
		parent := THIS^,
		fixture := _Fixture,
		scenario := COLLECTIONS_CONTRACT_SCENARIO.SORT_FAILURE_PRESERVES_ENTRIES
	);
	_QueueValidationAndGrowth : CollectionsContractTestCase(
		name := "QueueValidationAndGrowth",
		parent := THIS^,
		fixture := _Fixture,
		scenario := COLLECTIONS_CONTRACT_SCENARIO.QUEUE_VALIDATION_AND_GROWTH
	);
	_HashCollisionGrowth : CollectionsContractTestCase(
		name := "HashCollisionGrowth",
		parent := THIS^,
		fixture := _Fixture,
		scenario := COLLECTIONS_CONTRACT_SCENARIO.HASH_COLLISION_GROWTH
	);
	_HashEqualityRepresentations : CollectionsContractTestCase(
		name := "HashEqualityRepresentations",
		parent := THIS^,
		fixture := _Fixture,
		scenario := COLLECTIONS_CONTRACT_SCENARIO.HASH_EQUALITY_REPRESENTATIONS
	);
	_HashOwnershipAliases : CollectionsContractTestCase(
		name := "HashOwnershipAliases",
		parent := THIS^,
		fixture := _Fixture,
		scenario := COLLECTIONS_CONTRACT_SCENARIO.HASH_OWNERSHIP_ALIASES
	);
	_FullStaticDuplicateUpdates : CollectionsContractTestCase(
		name := "FullStaticDuplicateUpdates",
		parent := THIS^,
		fixture := _Fixture,
		scenario := COLLECTIONS_CONTRACT_SCENARIO.FULL_STATIC_DUPLICATE_UPDATES
	);
	_QueryFailureCleanup : CollectionsContractTestCase(
		name := "QueryFailureCleanup",
		parent := THIS^,
		fixture := _Fixture,
		scenario := COLLECTIONS_CONTRACT_SCENARIO.QUERY_FAILURE_CLEANUP
	);
	_ContainsCollectionCallbackFailures : CollectionsContractTestCase(
		name := "ContainsCollectionCallbackFailures",
		parent := THIS^,
		fixture := _Fixture,
		scenario := COLLECTIONS_CONTRACT_SCENARIO.CONTAINS_COLLECTION_CALLBACK_FAILURES
	);
	_GenericQueryReleaseMatrix : CollectionsContractTestCase(
		name := "GenericQueryReleaseMatrix",
		parent := THIS^,
		fixture := _Fixture,
		scenario := COLLECTIONS_CONTRACT_SCENARIO.GENERIC_QUERY_RELEASE_MATRIX
	);
	_AllCursorContracts : CollectionsContractTestCase(
		name := "AllCursorContracts",
		parent := THIS^,
		fixture := _Fixture,
		scenario := COLLECTIONS_CONTRACT_SCENARIO.ALL_CURSOR_CONTRACTS
	);
	_FixtureCleanupAfterException : CollectionsContractTestCase(
		name := "FixtureCleanupAfterException",
		parent := THIS^,
		fixture := _Fixture,
		scenario := COLLECTIONS_CONTRACT_SCENARIO.FIXTURE_CLEANUP_AFTER_EXCEPTION
	);
	_DefaultSortNumericBranches : CollectionsContractTestCase(
		name := "DefaultSortNumericBranches",
		parent := THIS^,
		fixture := _Fixture,
		scenario := COLLECTIONS_CONTRACT_SCENARIO.DEFAULT_SORT_NUMERIC_BRANCHES
	);
	_DefaultSortTextAndObjects : CollectionsContractTestCase(
		name := "DefaultSortTextAndObjects",
		parent := THIS^,
		fixture := _Fixture,
		scenario := COLLECTIONS_CONTRACT_SCENARIO.DEFAULT_SORT_TEXT_AND_OBJECTS
	);
	_DefaultSortExplicitAndRejection : CollectionsContractTestCase(
		name := "DefaultSortExplicitAndRejection",
		parent := THIS^,
		fixture := _Fixture,
		scenario := COLLECTIONS_CONTRACT_SCENARIO.DEFAULT_SORT_EXPLICIT_AND_REJECTION
	);
	_MissingCursorSources : CollectionsContractTestCase(
		name := "MissingCursorSources",
		parent := THIS^,
		fixture := _Fixture,
		scenario := COLLECTIONS_CONTRACT_SCENARIO.MISSING_CURSOR_SOURCES
	);

	_Children : ARRAY [0.._ChildCount - 1] OF TOF_Testing.ITestElement :=
	[
		_CopyFailurePreservesException,
		_SecondCopyFailureCleanup,
		_StaticFullCopyCleanup,
		_ByteOverlapAndBounds,
		_ByteSizeRejections,
		_ListOwnershipReplacement,
		_ListRemovalLimits,
		_SortFailurePreservesEntries,
		_QueueValidationAndGrowth,
		_HashCollisionGrowth,
		_HashEqualityRepresentations,
		_HashOwnershipAliases,
		_FullStaticDuplicateUpdates,
		_QueryFailureCleanup,
		_ContainsCollectionCallbackFailures,
		_GenericQueryReleaseMatrix,
		_AllCursorContracts,
		_FixtureCleanupAfterException,
		_DefaultSortNumericBranches,
		_DefaultSortTextAndObjects,
		_DefaultSortExplicitAndRejection,
		_MissingCursorSources
	];
END_VAR

//! <summary>Borrows the fixed child array. Callers must not modify it.</summary>
{attribute 'monitoring' := 'call'}
PROPERTY Children : REFERENCE TO ARRAY [0.._ChildCount - 1] OF TOF_Testing.ITestElement
GET
Children REF= _Children;
END_GET
END_PROPERTY

//! <summary>Borrows the concrete class name. Callers must not modify it.</summary>
{attribute 'monitoring' := 'call'}
PROPERTY ClassName : REFERENCE TO STRING
GET
ClassName REF= _ClassName;
END_GET
END_PROPERTY

//! <summary>Borrows the compiler-initialized namespace name. Callers must not modify it.</summary>
{attribute 'monitoring' := 'call'}
PROPERTY NamespaceName : REFERENCE TO STRING
GET
NamespaceName REF= CurrentNamespace.Name;
END_GET
END_PROPERTY

//! <summary>Reports the concrete instance size in bytes.</summary>
{attribute 'monitoring' := 'call'}
PROPERTY SelfSize : ULINT
GET
SelfSize := XSIZEOF(THIS^);
END_GET
END_PROPERTY

END_FUNCTION_BLOCK

// ---- Tests/Collections/Contract/CollectionsContractTestFixture.TcPOU
(*
SPDX-FileCopyrightText: © 2026 Oleksandr Tiutyk <trofimich@gmail.com>
SPDX-License-Identifier: MIT
License: https://opensource.org/license/mit
*)

(*!
<summary>Owns the collections and resources used by the collection contract cases.</summary>
<description>
A test group owns this fixture at a stable address. Run one case at a time in the owner task.
FinishScenario clears resources before a result is published, including when ExecuteScenario raises.
The fixture also clears owned resources on destruction. Terminal allocation failures use the task boundary.
</description>
*)

{attribute 'no_assign'}
{attribute 'no_explicit_call' := 'do not call this function block directly'}
FUNCTION_BLOCK CollectionsContractTestFixture EXTENDS TOF_Core.Object
VAR_STAT
	_ClassName : STRING := __POUNAME();
END_VAR
VAR
	//! <summary>Borrows the running case assertion context until FinishScenario.</summary>
	_Assertions : REFERENCE TO TOF_Testing.Assertions;
	//! <summary>Latches observable disposal failures for the current case.</summary>
	_ReleaseFailed : BOOL;

	_Scalar : DINT := 1;
	_OtherScalar : DINT := 2;
	_MiddleScalar : DINT := 13;
	_SignedKey : LINT := 1;
	_UnsignedKey : UINT := 1;
	_ByteValues : ARRAY [0..2] OF BYTE := [0, 1, 255];
	_RealBits : TOF_Core.REAL_UNION;
	_LongRealBits : TOF_Core.LREAL_UNION;

	_SortSigned : LINT;
	_SortUnsigned : UINT;
	_SortReal : LREAL;
	_SortText : STRING(16) := 'b';
	_SortWideText : WSTRING(16) := "a";
	_FirstComparable : CollectionComparableProbe;
	_SecondComparable : CollectionComparableProbe;

	_NullByteCursor : TOF_Collections.ByteListEnumerator(list := 0);
	_NullListCursor : TOF_Collections.ListEnumerator(list := 0);
	_NullQueueCursor : TOF_Collections.QueueEnumerator(queue := 0);
	_NullStackCursor : TOF_Collections.StackEnumerator(stack := 0);
	_NullDictionaryCursor : TOF_Collections.DictionaryEnumerator(dictionary := 0);
	_NullSetCursor : TOF_Collections.UniqueDataSetEnumerator(uniqueSet := 0);
	_NullCursors : ARRAY [0..5] OF TOF_Core.IEnumerator;

	_CloneExitCount : UDINT;
	_CloneSource : CollectionCloneProbe;
	_FailingCloneSource : CollectionCloneProbe;
	_Validator : CollectionValidatorProbe;
	_Equality : CollectionEqualityProbe;
	_Predicate : CollectionPredicateProbe;
	_Comparer : CollectionComparerProbe;

	_Bytes : TOF_Collections.ByteList<0>;
	_StaticBytes : TOF_Collections.ByteList<8>;
	_List : TOF_Collections.List<0>(valueValidator := 0);
	_Queue : TOF_Collections.Queue<0>(valueValidator := _Validator);
	_Stack : TOF_Collections.Stack<0>(valueValidator := 0);
	_Dictionary : TOF_Collections.Dictionary<0>(keyValidator := 0, valueValidator := 0, keyEqualityComparer := 0);
	_Set : TOF_Collections.UniqueDataSet<0>(valueValidator := 0, valueEqualityComparer := 0);
	_CollisionDictionary : TOF_Collections.Dictionary<0>(
		keyValidator := 0,
		valueValidator := 0,
		keyEqualityComparer := _Equality
	);
	_CollisionSet : TOF_Collections.UniqueDataSet<0>(valueValidator := 0, valueEqualityComparer := _Equality);

	_RejectedList : TOF_Collections.List<1>(valueValidator := _Validator);
	_RejectedQueue : TOF_Collections.Queue<1>(valueValidator := _Validator);
	_RejectedStack : TOF_Collections.Stack<1>(valueValidator := _Validator);
	_RejectedDictionary : TOF_Collections.Dictionary<1>(
		keyValidator := 0,
		valueValidator := _Validator,
		keyEqualityComparer := 0
	);
	_RejectedSet : TOF_Collections.UniqueDataSet<1>(valueValidator := _Validator, valueEqualityComparer := 0);

	_FullList : TOF_Collections.List<1>(valueValidator := 0);
	_FullQueue : TOF_Collections.Queue<1>(valueValidator := 0);
	_FullStack : TOF_Collections.Stack<1>(valueValidator := 0);
	_FullDictionary : TOF_Collections.Dictionary<1>(keyValidator := 0, valueValidator := 0, keyEqualityComparer := 0);
	_FullSet : TOF_Collections.UniqueDataSet<1>(valueValidator := 0, valueEqualityComparer := 0);

	//! <summary>Retains unaccepted allocations and cursors across an aborted helper call.</summary>
	_OwnedObject : TOF_Core.IObject;
	_OwnedValue : TOF_Core.GENERIC_VALUE;
	_Query : TOF_Core.GENERIC_VALUE;
	_BorrowedSource : TOF_Core.GENERIC_VALUE;
	_Enumerator : TOF_Core.IEnumerator;
	_SecondEnumerator : TOF_Core.IEnumerator;
END_VAR

(*!
<summary>Runs one collection contract scenario using the active test assertions.</summary>
<description>
Starts with empty collections, reset probe injections and no retained resources. A scenario can raise an
unexpected exception. FinishScenario is required before publishing its result or starting another case.
</description>
<param name="scenario">Selected contract scenario.</param>
<param name="assertions">Context bound to the running test case.</param>
*)
METHOD INTERNAL ExecuteScenario
VAR_INPUT
	scenario : COLLECTIONS_CONTRACT_SCENARIO;
	assertions : REFERENCE TO TOF_Testing.Assertions;
END_VAR
_Assertions REF= assertions;
_ReleaseFailed := FALSE;
cleanupFixtures();
_CloneSource.ObserveExit(counter := _CloneExitCount);
_CloneSource.ClearCloneTransportOnExit := TRUE;
_CloneExitCount := TOF_Core.UnsignedInt32.ZERO;

CASE scenario OF
	COLLECTIONS_CONTRACT_SCENARIO.COPY_FAILURE_PRESERVES_EXCEPTION:
		copyFailurePreservesException();

	COLLECTIONS_CONTRACT_SCENARIO.SECOND_COPY_FAILURE_CLEANUP:
		secondCopyFailureCleanup();

	COLLECTIONS_CONTRACT_SCENARIO.STATIC_FULL_COPY_CLEANUP:
		staticFullCopyCleanup();

	COLLECTIONS_CONTRACT_SCENARIO.BYTE_OVERLAP_AND_BOUNDS:
		byteOverlapAndBounds();

	COLLECTIONS_CONTRACT_SCENARIO.BYTE_SIZE_REJECTIONS:
		byteSizeRejections();

	COLLECTIONS_CONTRACT_SCENARIO.LIST_OWNERSHIP_REPLACEMENT:
		listOwnershipReplacement();

	COLLECTIONS_CONTRACT_SCENARIO.LIST_REMOVAL_LIMITS:
		listRemovalLimits();

	COLLECTIONS_CONTRACT_SCENARIO.SORT_FAILURE_PRESERVES_ENTRIES:
		sortFailurePreservesEntries();

	COLLECTIONS_CONTRACT_SCENARIO.QUEUE_VALIDATION_AND_GROWTH:
		queueValidationAndGrowth();

	COLLECTIONS_CONTRACT_SCENARIO.HASH_COLLISION_GROWTH:
		hashCollisionGrowth();

	COLLECTIONS_CONTRACT_SCENARIO.HASH_EQUALITY_REPRESENTATIONS:
		hashEqualityRepresentations();

	COLLECTIONS_CONTRACT_SCENARIO.HASH_OWNERSHIP_ALIASES:
		hashOwnershipAliases();

	COLLECTIONS_CONTRACT_SCENARIO.FULL_STATIC_DUPLICATE_UPDATES:
		fullStaticDuplicateUpdates();

	COLLECTIONS_CONTRACT_SCENARIO.QUERY_FAILURE_CLEANUP:
		queryFailureCleanup();

	COLLECTIONS_CONTRACT_SCENARIO.CONTAINS_COLLECTION_CALLBACK_FAILURES:
		containsCollectionCallbackFailures();

	COLLECTIONS_CONTRACT_SCENARIO.GENERIC_QUERY_RELEASE_MATRIX:
		genericQueryReleaseMatrix();

	COLLECTIONS_CONTRACT_SCENARIO.ALL_CURSOR_CONTRACTS:
		allCursorContracts();

	COLLECTIONS_CONTRACT_SCENARIO.FIXTURE_CLEANUP_AFTER_EXCEPTION:
		fixtureCleanupAfterException();

	COLLECTIONS_CONTRACT_SCENARIO.DEFAULT_SORT_NUMERIC_BRANCHES:
		defaultSortNumericBranches();

	COLLECTIONS_CONTRACT_SCENARIO.DEFAULT_SORT_TEXT_AND_OBJECTS:
		defaultSortTextAndObjects();

	COLLECTIONS_CONTRACT_SCENARIO.DEFAULT_SORT_EXPLICIT_AND_REJECTION:
		defaultSortExplicitAndRejection();

	COLLECTIONS_CONTRACT_SCENARIO.MISSING_CURSOR_SOURCES:
		missingCursorSources();
ELSE
	_Assertions.ThatBool(
		actual := FALSE,
		message := "Invalid collection contract scenario"
	).IsTrue();
END_CASE
END_METHOD

(*!
<summary>Clears the fixture and returns whether checked releases succeeded.</summary>
<description>
Detaches the assertion context before cleanup. Returns FALSE for a failed cursor or interface release
observed during the case or teardown. Generic-value Release remains best effort.
</description>
*)
METHOD INTERNAL FinishScenario : BOOL
_Assertions REF= 0;
cleanupFixtures();
FinishScenario := NOT _ReleaseFailed;
END_METHOD

(*!
<summary>Checks independent cursors, generic byte values, Reset and repeated exhaustion for six containers.</summary>
<description>
Starts with independent fixture state. The harness clears persistent resources before publication, including
after an aborted call. Terminal OOM injection is reserved for an isolated test.
</description>
*)
METHOD PRIVATE allCursorContracts
VAR
	i : DINT;
END_VAR
_Bytes.AppendData(data := ADR(_ByteValues), dataSize := 3);
_List.AppendCopy(value := _Scalar);
_Queue.EnqueueCopy(value := _Scalar);
_Stack.PushCopy(value := _Scalar);
_Dictionary.SetCopy(key := _Scalar, value := _OtherScalar);
_Set.SetCopy(value := _Scalar);
checkCursor(source := _Bytes);
checkCursor(source := _List);
checkCursor(source := _Queue);
checkCursor(source := _Stack);
checkCursor(source := _Dictionary);
checkCursor(source := _Set);

_Enumerator := _Bytes.CreateEnumerator();
_Assertions.ThatBool(
	actual := _Enumerator <> 0,
	message := "Byte list must create a cursor"
).IsTrue();

IF _Enumerator = 0 THEN
	RETURN;
END_IF

FOR i := 0 TO 2 DO
	_Assertions.ThatBool(
		actual := _Enumerator.MoveNext(),
		message := "Byte cursor must visit every byte"
	).IsTrue();
	_Assertions.ThatByte(
		actual := _Enumerator.Current.AsByte(),
		message := "Generic Current must address cached byte storage, including zero"
	).ToBe(expected := _ByteValues[i]);
END_FOR

releaseCursors();
_Bytes.Clear();
_List.Clear();
_Queue.Clear();
_Stack.Clear();
_Dictionary.Clear();
_Set.Clear();
checkCursor(source := _Bytes);
checkCursor(source := _List);
checkCursor(source := _Queue);
checkCursor(source := _Stack);
checkCursor(source := _Dictionary);
checkCursor(source := _Set);
END_METHOD

(*!
<summary>Checks a caught framework failure after resource cleanup.</summary>
<description>
Captures and consumes the exception within the current call; no exception interface survives task cleanup.
</description>
*)
METHOD PRIVATE assertOriginalFailure
VAR_INPUT
	exceptionCode : __SYSTEM.ExceptionCode;
	expectedMessage : WSTRING;
END_VAR
VAR
	caughtException : TOF_Core.IException;
	standardException : TOF_Core.IStandardException;
	actualMessage : TOF_Core.ERROR_MESSAGE;
END_VAR
caughtException := TOF_Core.ExceptionManager.GetLastException(
	exceptionCode := exceptionCode,
	catchPointNamespaceName := NamespaceName,
	catchPointPOUName := __POUNAME(),
	catchPointPosition := __POSITION()
);
_Assertions.ThatBool(
	actual := __QUERYINTERFACE(caughtException, standardException),
	message := "Original StandardException category must be preserved"
).IsTrue();
IF standardException = 0 THEN
	RETURN;
END_IF

actualMessage := caughtException.GetMessage();
_Assertions.That(
	actual := actualMessage,
	message := "Original message must survive"
).ToBe(expected := expectedMessage);
END_METHOD

(*!
<summary>Supports byte self-growth, overlapping loads, empty removal and checked ranges.</summary>
<description>
Starts with independent fixture state. The harness clears persistent resources before publication, including
after an aborted call. Terminal OOM injection is reserved for an isolated test.
</description>
*)
METHOD PRIVATE byteOverlapAndBounds
VAR
	i : DINT;
END_VAR
_Bytes.Remove(value := 7);
_StaticBytes.Remove(value := 7);
_Bytes.AppendData(data := ADR(_ByteValues), dataSize := 3);
_Bytes.AppendData(data := _Bytes.DataAddress, dataSize := _Bytes.Length);
_Assertions.ThatDInt(
	actual := _Bytes.Length,
	message := "Self-append must grow to six bytes"
).ToBe(expected := 6);

FOR i := 0 TO 5 DO
	_Assertions.ThatByte(
		actual := _Bytes.Get(index := i),
		message := "Self-growth must retain the source bytes"
	).ToBe(expected := _ByteValues[i MOD 3]);
END_FOR

_Bytes.LoadFromData(data := _Bytes.DataAddress + 1, dataSize := 4, startIndex := 0);
_Assertions.ThatDInt(
	actual := _Bytes.Length,
	message := "Overlapping load must truncate the tail"
).ToBe(expected := 4);
_Assertions.ThatByte(
	actual := _Bytes.Get(index := 0),
	message := "Overlap must copy the old second byte"
).ToBe(expected := 1);
_Assertions.ThatByte(
	actual := _Bytes.Get(index := 1),
	message := "Overlap must preserve byte 255"
).ToBe(expected := 255);
_Bytes.LoadFromData(data := 0, dataSize := 0, startIndex := 2);
_Assertions.ThatDInt(
	actual := _Bytes.Length,
	message := "Null zero load must preserve Length"
).ToBe(expected := 4);
_Bytes.Clear(releaseDynamicMemory := TRUE);
_Assertions.ThatDInt(
	actual := _Bytes.Capacity,
	message := "Explicit release must drop byte capacity"
).ToBe(expected := 0);

_StaticBytes.AppendData(data := ADR(_ByteValues), dataSize := 3);
_StaticBytes.AppendData(data := _StaticBytes.DataAddress, dataSize := 3);
_StaticBytes.LoadFromData(data := _StaticBytes.DataAddress + 1, dataSize := 4, startIndex := 0);
_Assertions.ThatByte(
	actual := _StaticBytes.Get(index := 0),
	message := "Static overlap must be supported"
).ToBe(expected := 1);
_StaticBytes.RemoveAt(index := 1, count := 0);
_Assertions.ThatDInt(
	actual := _StaticBytes.Length,
	message := "Validated zero removal must be a no-op"
).ToBe(expected := 4);
END_METHOD

(*!
<summary>Rejects oversized generic byte ranges and overflowing end positions before reading input.</summary>
<description>
Starts with independent fixture state. The harness clears persistent resources before publication, including
after an aborted call. Terminal OOM injection is reserved for an isolated test.
</description>
*)
METHOD PRIVATE byteSizeRejections
VAR
	i : DINT;
	rejected : BOOL;
	exceptionCode : __SYSTEM.ExceptionCode;
	caughtException : TOF_Core.IException;
	rangeException : TOF_Core.IArgumentOutOfRangeException;
END_VAR
_Bytes.AppendData(data := ADR(_ByteValues), dataSize := 3);
_Query := TOF_Core.GenericValueFactory.FromParts(
	genericTypeClass := TOF_Core.GENERIC_TYPE_CLASS.UINT_8,
	address := ADR(_ByteValues),
	size := TO_ULINT(TOF_Core.SignedInt32.MAX_VALUE) + 1,
	memoryManagementBehavior := TOF_Core.GENERIC_MEMORY_MANAGEMENT_BEHAVIOR.STORE_ORIGINAL_REFERENCE_AND_NOT_OWNS_MEMORY
);

FOR i := 0 TO 3 DO
	rejected := FALSE;

	__TRY
		CASE i OF
			0:
				_Bytes.AppendGeneric(data := _Query);
			1:
				_Bytes.LoadFromGeneric(data := _Query);
			2:
				_Bytes.AppendData(data := ADR(_ByteValues), dataSize := TOF_Core.SignedInt32.MAX_VALUE);
			3:
				_Bytes.RemoveAt(index := 1, count := TOF_Core.SignedInt32.MAX_VALUE);
		END_CASE
	__CATCH(exceptionCode)
		rejected := TRUE;
		caughtException := TOF_Core.ExceptionManager.GetLastException(
			exceptionCode := exceptionCode,
			catchPointNamespaceName := NamespaceName,
			catchPointPOUName := __POUNAME(),
			catchPointPosition := __POSITION()
		);
		_Assertions.ThatBool(
			actual := __QUERYINTERFACE(caughtException, rangeException),
			message := "Oversized byte range must report ArgumentOutOfRangeException"
		).IsTrue();
	__ENDTRY

	_Assertions.ThatBool(
		actual := rejected,
		message := "Oversized byte request must be rejected"
	).IsTrue();
	_Assertions.ThatDInt(
		actual := _Bytes.Length,
		message := "Rejected range must preserve Length"
	).ToBe(expected := 3);
	_Assertions.ThatByte(
		actual := _Bytes.Get(index := 2),
		message := "Rejected range must preserve bytes"
	).ToBe(expected := 255);
END_FOR

_Query.Reset();
END_METHOD

(*!
<summary>Checks traversal and invalid-current states without changing the borrowed source.</summary>
<description>
The source stays alive and structurally unchanged. Cursor ownership remains in fixture fields if a call raises.
</description>
*)
METHOD PRIVATE checkCursor
VAR_INPUT
	source : TOF_Collections.ICollection;
END_VAR
VAR
	i : DINT;
END_VAR
_Enumerator := source.CreateEnumerator();
_SecondEnumerator := source.CreateEnumerator();

_Assertions.ThatBool(
	actual := _Enumerator <> 0 AND_THEN _SecondEnumerator <> 0,
	message := "Each traversal must create a cursor"
).IsTrue();

IF _Enumerator = 0 OR_ELSE _SecondEnumerator = 0 THEN
	releaseCursors();

	RETURN;
END_IF

_Assertions.ThatBool(
	actual := _Enumerator <> _SecondEnumerator,
	message := "Owned cursors must be independent"
).IsTrue();

IF _Enumerator = _SecondEnumerator THEN
	releaseCursors();

	RETURN;
END_IF

_Assertions.ThatBool(
	actual := _Enumerator.Current.IsNull,
	message := "Current before MoveNext must be empty"
).IsTrue();

FOR i := 0 TO source.Length - 1 DO
	_Assertions.ThatBool(
		actual := _Enumerator.MoveNext(),
		message := "Cursor must visit every source entry"
	).IsTrue();
	_Assertions.ThatBool(
		actual := _Enumerator.Current.IsNull,
		message := "Current must expose the visited entry"
	).IsFalse();
END_FOR

_Assertions.ThatBool(
	actual := _Enumerator.MoveNext(),
	message := "Cursor must stop at source end"
).IsFalse();
_Assertions.ThatBool(
	actual := _Enumerator.MoveNext(),
	message := "Exhausted cursor must stay exhausted"
).IsFalse();
_Assertions.ThatBool(
	actual := _Enumerator.Current.IsNull,
	message := "Current after exhaustion must be empty"
).IsTrue();
_Assertions.ThatBool(
	actual := _SecondEnumerator.MoveNext(),
	message := "Second cursor must retain an independent position"
).ToBe(expected := source.Length > TOF_Core.SignedInt32.ZERO);
_Enumerator.Reset();
_Assertions.ThatBool(
	actual := _Enumerator.Current.IsNull,
	message := "Current after Reset must be empty"
).IsTrue();
_Assertions.ThatBool(
	actual := _Enumerator.MoveNext(),
	message := "Reset must restore the initial cursor position"
).ToBe(expected := source.Length > TOF_Core.SignedInt32.ZERO);
releaseCursors();
END_METHOD

(*!
<summary>Clears all fixture-owned resources and resets the injected failures.</summary>
<description>
Uses non-allocating, non-throwing release paths. All probe counters and borrowed source values are persistent.
</description>
*)
METHOD PRIVATE cleanupFixtures
releaseCursors();
_CloneSource.ThrowOnEquality := FALSE;
_FailingCloneSource.ThrowOnClone := FALSE;
_Validator.Reject := FALSE;
_Equality.ThrowOnHash := FALSE;
_Equality.ThrowOnEquality := FALSE;
_Predicate.ThrowOnCall := 0;
_Comparer.ThrowOnCall := 0;

_Bytes.Clear(releaseDynamicMemory := TRUE);
_StaticBytes.Clear(releaseDynamicMemory := TRUE);
_List.Clear();
_Queue.Clear();
_Stack.Clear();
_Dictionary.Clear();
_Set.Clear();
_CollisionDictionary.Clear();
_CollisionSet.Clear();
_Equality.MatchEveryValue := FALSE;
_RejectedList.Clear();
_RejectedQueue.Clear();
_RejectedStack.Clear();
_RejectedDictionary.Clear();
_RejectedSet.Clear();
_FullList.Clear();
_FullQueue.Clear();
_FullStack.Clear();
_FullDictionary.Clear();
_FullSet.Clear();

_OwnedValue.Release();
_Query.Release();
_BorrowedSource.Reset();

IF _OwnedObject <> 0 THEN
	IF NOT TOF_Core.Memory.TryReleaseDynamicObject(instance := _OwnedObject) THEN
		_ReleaseFailed := TRUE;
	END_IF
END_IF
END_METHOD

(*!
<summary>Preserves the original validator failure across cleanup in all seven Copy methods.</summary>
<description>
Starts with independent fixture state. The harness clears persistent resources before publication, including
after an aborted call. Terminal OOM injection is reserved for an isolated test.
</description>
*)
METHOD PRIVATE copyFailurePreservesException
VAR
	rejected : BOOL;
	exceptionCode : __SYSTEM.ExceptionCode;
END_VAR
_RejectedList.AppendCopy(value := _Scalar);
_Validator.Reject := TRUE;

rejected := FALSE;
_CloneExitCount := TOF_Core.UnsignedInt32.ZERO;

__TRY
	_RejectedList.AppendCopy(value := _CloneSource, isObject := TRUE);
__CATCH(exceptionCode)
	rejected := TRUE;
	assertOriginalFailure(exceptionCode := exceptionCode, expectedMessage := "Collection validation rejected");
__ENDTRY

_Assertions.ThatBool(
	actual := rejected,
	message := "Failure must propagate"
).IsTrue();
_Assertions.ThatUDInt(
	actual := _CloneExitCount,
	message := "Owned temporary must be released exactly once"
).ToBe(expected := 1);

rejected := FALSE;
_CloneExitCount := TOF_Core.UnsignedInt32.ZERO;

__TRY
	_RejectedList.InsertCopy(index := 0, value := _CloneSource, isObject := TRUE);
__CATCH(exceptionCode)
	rejected := TRUE;
	assertOriginalFailure(exceptionCode := exceptionCode, expectedMessage := "Collection validation rejected");
__ENDTRY

_Assertions.ThatBool(
	actual := rejected,
	message := "Failure must propagate"
).IsTrue();
_Assertions.ThatUDInt(
	actual := _CloneExitCount,
	message := "Owned temporary must be released exactly once"
).ToBe(expected := 1);

rejected := FALSE;
_CloneExitCount := TOF_Core.UnsignedInt32.ZERO;

__TRY
	_RejectedList.SetCopy(index := 0, value := _CloneSource, isObject := TRUE);
__CATCH(exceptionCode)
	rejected := TRUE;
	assertOriginalFailure(exceptionCode := exceptionCode, expectedMessage := "Collection validation rejected");
__ENDTRY

_Assertions.ThatBool(
	actual := rejected,
	message := "Failure must propagate"
).IsTrue();
_Assertions.ThatUDInt(
	actual := _CloneExitCount,
	message := "Owned temporary must be released exactly once"
).ToBe(expected := 1);

rejected := FALSE;
_CloneExitCount := TOF_Core.UnsignedInt32.ZERO;

__TRY
	_RejectedQueue.EnqueueCopy(value := _CloneSource, isObject := TRUE);
__CATCH(exceptionCode)
	rejected := TRUE;
	assertOriginalFailure(exceptionCode := exceptionCode, expectedMessage := "Collection validation rejected");
__ENDTRY

_Assertions.ThatBool(
	actual := rejected,
	message := "Failure must propagate"
).IsTrue();
_Assertions.ThatUDInt(
	actual := _CloneExitCount,
	message := "Owned temporary must be released exactly once"
).ToBe(expected := 1);

rejected := FALSE;
_CloneExitCount := TOF_Core.UnsignedInt32.ZERO;

__TRY
	_RejectedStack.PushCopy(value := _CloneSource, isObject := TRUE);
__CATCH(exceptionCode)
	rejected := TRUE;
	assertOriginalFailure(exceptionCode := exceptionCode, expectedMessage := "Collection validation rejected");
__ENDTRY

_Assertions.ThatBool(
	actual := rejected,
	message := "Failure must propagate"
).IsTrue();
_Assertions.ThatUDInt(
	actual := _CloneExitCount,
	message := "Owned temporary must be released exactly once"
).ToBe(expected := 1);

rejected := FALSE;
_CloneExitCount := TOF_Core.UnsignedInt32.ZERO;

__TRY
	_RejectedDictionary.SetCopy(key := _Scalar, value := _CloneSource, valueIsObject := TRUE);
__CATCH(exceptionCode)
	rejected := TRUE;
	assertOriginalFailure(exceptionCode := exceptionCode, expectedMessage := "Collection validation rejected");
__ENDTRY

_Assertions.ThatBool(
	actual := rejected,
	message := "Failure must propagate"
).IsTrue();
_Assertions.ThatUDInt(
	actual := _CloneExitCount,
	message := "Owned temporary must be released exactly once"
).ToBe(expected := 1);

rejected := FALSE;
_CloneExitCount := TOF_Core.UnsignedInt32.ZERO;

__TRY
	_RejectedSet.SetCopy(value := _CloneSource, isObject := TRUE);
__CATCH(exceptionCode)
	rejected := TRUE;
	assertOriginalFailure(exceptionCode := exceptionCode, expectedMessage := "Collection validation rejected");
__ENDTRY

_Assertions.ThatBool(
	actual := rejected,
	message := "Failure must propagate"
).IsTrue();
_Assertions.ThatUDInt(
	actual := _CloneExitCount,
	message := "Owned temporary must be released exactly once"
).ToBe(expected := 1);

_Assertions.ThatDInt(
	actual := _RejectedList.Length,
	message := "Rejected replacement must retain entry"
).ToBe(expected := 1);
_Assertions.ThatDInt(
	actual := _RejectedList.Get(index := 0).AsDInt(),
	message := "Entry must survive"
).ToBe(expected := _Scalar);
_Assertions.ThatBool(
	actual := _RejectedQueue.Empty,
	message := "Rejected queue must remain empty"
).IsTrue();
_Assertions.ThatBool(
	actual := _RejectedStack.Empty,
	message := "Rejected stack must remain empty"
).IsTrue();
_Assertions.ThatBool(
	actual := _RejectedDictionary.Empty,
	message := "Rejected dictionary must remain empty"
).IsTrue();
_Assertions.ThatBool(
	actual := _RejectedSet.Empty,
	message := "Rejected set must remain empty"
).IsTrue();
END_METHOD

(*!
<summary>Preserves explicit comparer priority and reports unsupported default pairs without losing entries.</summary>
<description>
Uses persistent collection and source fixtures. Each case prepares an independent initial state;
comparison failures retain descriptors without promising rollback of completed swaps.
</description>
*)
METHOD PRIVATE defaultSortExplicitAndRejection
VAR
	rejected : BOOL;
	exceptionCode : __SYSTEM.ExceptionCode;
	caughtException : TOF_Core.IException;
	conversionException : TOF_Core.IGenericConversionNotSupportedException;
	objectValue : TOF_Core.GENERIC_VALUE;
END_VAR
_Comparer.ResetCount();
_Comparer.ThrowOnCall := 1;
_List.Sort();
_List.Sort(comparer := _Comparer);
_List.AppendCopy(value := _Scalar);
_List.Sort();
_List.Sort(comparer := _Comparer);
_Assertions.ThatUDInt(
	actual := _Comparer.CallCount,
	message := "Empty and singleton sort must not compare"
).ToBe(expected := 0);
_List.AppendCopy(value := _SortText);

__TRY
	_List.Sort(comparer := _Comparer);
__CATCH(exceptionCode)
	rejected := TRUE;
	assertOriginalFailure(exceptionCode := exceptionCode, expectedMessage := "Collection comparer rejected");
__ENDTRY

_Assertions.ThatBool(
	actual := rejected,
	message := "Explicit comparer must run before default compatibility checks"
).IsTrue();
_Assertions.ThatUDInt(
	actual := _Comparer.CallCount,
	message := "Explicit comparer must receive the pair"
).ToBe(expected := 1);
rejected := FALSE;

__TRY
	_List.Sort();
__CATCH(exceptionCode)
	rejected := TRUE;
	caughtException := TOF_Core.ExceptionManager.GetLastException(
		exceptionCode := exceptionCode,
		catchPointNamespaceName := NamespaceName,
		catchPointPOUName := __POUNAME(),
		catchPointPosition := __POSITION()
	);
	_Assertions.ThatBool(
		actual := __QUERYINTERFACE(caughtException, conversionException),
		message := "Unsupported default order must report GenericConversionNotSupportedException"
	).IsTrue();
__ENDTRY

_Assertions.ThatBool(
	actual := rejected,
	message := "Incompatible numeric and text values must reject default sorting"
).IsTrue();
_Assertions.ThatDInt(
	actual := _List.Length,
	message := "Default rejection must retain all entries"
).ToBe(expected := 2);
_Assertions.ThatBool(
	actual := _List.Get(index := 0).IsMemoryOwner,
	message := "Default rejection must retain first owner"
).IsTrue();
_Assertions.ThatBool(
	actual := _List.Get(index := 1).IsMemoryOwner,
	message := "Default rejection must retain second owner"
).IsTrue();
_List.Clear();
objectValue := TOF_Core.GenericValueFactory.FromAnyType(
	value := _CloneSource,
	isObject := TRUE,
	memoryManagementBehavior := TOF_Core.GENERIC_MEMORY_MANAGEMENT_BEHAVIOR.STORE_ORIGINAL_REFERENCE_AND_NOT_OWNS_MEMORY
);
_List.AppendGeneric(value := objectValue);
_List.Sort();
_List.AppendGeneric(value := objectValue);
rejected := FALSE;

__TRY
	_List.Sort();
__CATCH(exceptionCode)
	rejected := TRUE;
	caughtException := TOF_Core.ExceptionManager.GetLastException(
		exceptionCode := exceptionCode,
		catchPointNamespaceName := NamespaceName,
		catchPointPOUName := __POUNAME(),
		catchPointPosition := __POSITION()
	);
	_Assertions.ThatBool(
		actual := __QUERYINTERFACE(caughtException, conversionException),
		message := "Unsupported default order must report GenericConversionNotSupportedException"
	).IsTrue();
__ENDTRY

_Assertions.ThatBool(
	actual := rejected,
	message := "OBJECT default order requires IComparable"
).IsTrue();
_Assertions.ThatDInt(
	actual := _List.Length,
	message := "Unsupported OBJECT sorting must retain descriptors"
).ToBe(expected := 2);
END_METHOD

(*!
<summary>Sorts mixed numeric representations with omitted or null comparer in both algorithm branches.</summary>
<description>
Uses persistent collection and source fixtures. Each case prepares an independent initial state;
comparison failures retain descriptors without promising rollback of completed swaps.
</description>
*)
METHOD PRIVATE defaultSortNumericBranches
VAR
	i : DINT;
	count : DINT;
	expectedValue : DINT;
	expectedDescriptor : TOF_Core.GENERIC_VALUE;
	sortView : TOF_Collections.IList;
END_VAR
sortView := _List;

FOR count := 16 TO 17 DO
	_List.Clear();

	FOR i := count TO 1 BY -1 DO
		CASE i MOD 3 OF
			0:
				_SortReal := TO_LREAL(i);
				_List.AppendCopy(value := _SortReal);
			1:
				_SortSigned := TO_LINT(i);
				_List.AppendCopy(value := _SortSigned);
			2:
				_SortUnsigned := TO_UINT(i);
				_List.AppendCopy(value := _SortUnsigned);
		END_CASE
	END_FOR

	sortView.Sort();

	FOR i := 0 TO count - 1 DO
		expectedValue := i + 1;
		expectedDescriptor := TOF_Core.GenericValueFactory.FromDIntReference(value := expectedValue);
		_Assertions.ThatBool(
			actual := _List.Get(index := i).CompareTo(otherValue := expectedDescriptor)
				= TOF_Core.COMPARISON_RESULT.FIRST_EQUAL_TO_SECOND,
			message := "Default ascending order must compare mixed numeric values by value"
		).IsTrue();
	END_FOR

	_List.Sort(comparer := 0, direction := TOF_Core.SORT_DIRECTION.DESCENDING);

	FOR i := 0 TO count - 1 DO
		expectedValue := count - i;
		expectedDescriptor := TOF_Core.GenericValueFactory.FromDIntReference(value := expectedValue);
		_Assertions.ThatBool(
			actual := _List.Get(index := i).CompareTo(otherValue := expectedDescriptor)
				= TOF_Core.COMPARISON_RESULT.FIRST_EQUAL_TO_SECOND,
			message := "Null comparer must select the same default order in descending sorting"
		).IsTrue();
		_Assertions.ThatBool(
			actual := _List.Get(index := i).IsMemoryOwner,
			message := "Default sorting must retain owners"
		).IsTrue();
	END_FOR
END_FOR
END_METHOD

(*!
<summary>Uses natural mixed-text and IComparable OBJECT ordering without catalogue selection.</summary>
<description>
Uses persistent collection and source fixtures. Each case prepares an independent initial state;
comparison failures retain descriptors without promising rollback of completed swaps.
</description>
*)
METHOD PRIVATE defaultSortTextAndObjects
VAR
	objectValue : TOF_Core.GENERIC_VALUE;
END_VAR
_List.AppendCopy(value := _SortText);
_List.AppendCopy(value := _SortWideText);
_List.Sort();
_Assertions.ThatWideString(
	actual := _List.Get(index := 0).AsWString255(),
	message := "Default sort must compare mixed STRING and WSTRING text"
).ToBe(expected := "a");
_Assertions.ThatWideString(
	actual := _List.Get(index := 1).AsWString255(),
	message := "Default mixed-text order must retain the second value"
).ToBe(expected := "b");
_List.Clear();
_FirstComparable.SortValue := 2;
_SecondComparable.SortValue := 1;
objectValue := TOF_Core.GenericValueFactory.FromAnyType(
	value := _FirstComparable,
	isObject := TRUE,
	memoryManagementBehavior := TOF_Core.GENERIC_MEMORY_MANAGEMENT_BEHAVIOR.STORE_ORIGINAL_REFERENCE_AND_NOT_OWNS_MEMORY
);
_List.AppendGeneric(value := objectValue);
objectValue := TOF_Core.GenericValueFactory.FromAnyType(
	value := _SecondComparable,
	isObject := TRUE,
	memoryManagementBehavior := TOF_Core.GENERIC_MEMORY_MANAGEMENT_BEHAVIOR.STORE_ORIGINAL_REFERENCE_AND_NOT_OWNS_MEMORY
);
_List.AppendGeneric(value := objectValue);
_List.Sort();
_Assertions.ThatBool(
	actual := TO_LWORD(_List.Get(index := 0).Address) = TO_LWORD(_SecondComparable.SelfAddress),
	message := "Default OBJECT ordering must invoke IComparable"
).IsTrue();
_Assertions.ThatBool(
	actual := _List.Get(index := 0).IsMemoryOwner,
	message := "Borrowed OBJECT must remain borrowed"
).IsFalse();
END_METHOD

(*!
<summary>Releases persistent resources during fixture destruction without allocating or raising.</summary>
*)
METHOD FB_exit : BOOL
VAR_INPUT
	bInCopyCode : BOOL;
END_VAR
cleanupFixtures();
END_METHOD

(*!
<summary>Retains resources through an intermediate throwing call and cleans them explicitly afterwards.</summary>
<description>
Starts with independent fixture state. The harness clears persistent resources before publication, including
after an aborted call. Terminal OOM injection is reserved for an isolated test.
</description>
*)
METHOD PRIVATE fixtureCleanupAfterException
VAR
	rejected : BOOL;
	exceptionCode : __SYSTEM.ExceptionCode;
END_VAR
_List.AppendCopy(value := _Scalar);

__TRY
	prepareResourcesThenReject();
__CATCH(exceptionCode)
	rejected := TRUE;
	assertOriginalFailure(exceptionCode := exceptionCode, expectedMessage := "Collection fixture rejected");
__ENDTRY

_Assertions.ThatBool(
	actual := rejected,
	message := "Fixture injection must reach the local handler"
).IsTrue();
_Assertions.ThatBool(
	actual := _Enumerator <> 0,
	message := "Cursor ownership must survive the aborted helper"
).IsTrue();
_Assertions.ThatBool(
	actual := _OwnedValue.IsMemoryOwner,
	message := "Payload ownership must survive the aborted helper"
).IsTrue();
releaseCursors();
_Assertions.ThatBool(
	actual := _Enumerator = 0,
	message := "Cursor alias must be reset after cleanup"
).IsTrue();
_OwnedValue.Release();
_Assertions.ThatUDInt(
	actual := _CloneExitCount,
	message := "Retained probe must be destroyed once"
).ToBe(expected := 1);
_Assertions.ThatDInt(
	actual := _List.Length,
	message := "Cursor disposal must not dispose its source"
).ToBe(expected := 1);
END_METHOD

(*!
<summary>Updates equal entries in full static hash containers without adding a slot.</summary>
<description>
Starts with independent fixture state. The harness clears persistent resources before publication, including
after an aborted call. Terminal OOM injection is reserved for an isolated test.
</description>
*)
METHOD PRIVATE fullStaticDuplicateUpdates
VAR
	keyAddress : PVOID;
END_VAR
_FullDictionary.SetCopy(key := _Scalar, value := _Scalar);
_FullSet.SetCopy(value := _Scalar);
keyAddress := _FullDictionary.GetKeyValuePairByIndex(index := 0).Key.Address;
_FullDictionary.SetCopy(key := _Scalar, value := _OtherScalar);
_FullSet.SetCopy(value := _Scalar);
_Assertions.ThatDInt(
	actual := _FullDictionary.Length,
	message := "Duplicate update must not need a slot"
).ToBe(expected := 1);
_Assertions.ThatDInt(
	actual := _FullSet.Length,
	message := "Duplicate set replacement must not need a slot"
).ToBe(expected := 1);
_Assertions.ThatBool(
	actual := keyAddress = _FullDictionary.GetKeyValuePairByIndex(index := 0).Key.Address,
	message := "Dictionary must retain its existing equal key allocation"
).IsTrue();
_Assertions.ThatDInt(
	actual := _FullDictionary.GetKeyValuePairByIndex(index := 0).Value.AsDInt(),
	message := "Full dictionary must accept the replacement value"
).ToBe(expected := _OtherScalar);
END_METHOD

(*!
<summary>Checks found/missing queries with owned/borrowed payload and explicit release on/off.</summary>
<description>
Exercises seven generic dictionary/set queries over 56 combinations. Universal fixture equality permits
an owned query to match without aliasing any retained allocation. The source counter is persistent and
cleanup never dereferences a caller alias after requested release.
</description>
*)
METHOD PRIVATE genericQueryReleaseMatrix
VAR
	foundCase : DINT;
	ownedCase : DINT;
	releaseCase : DINT;
	operation : DINT;
	position : DINT;
	found : BOOL;
	releaseQuery : BOOL;
	foundValue : TOF_Core.GENERIC_VALUE;
	queryAsInterface : TOF_Core.IObject;
	queryForCall : TOF_Core.GENERIC_VALUE;
	scenarioDescription : WSTRING(255);
END_VAR
_CloneSource.ObserveExit(counter := _CloneExitCount);
_CloneSource.ClearCloneTransportOnExit := TRUE;
_Equality.MatchEveryValue := TRUE;

FOR foundCase := 0 TO 1 DO
	FOR ownedCase := 0 TO 1 DO
		FOR releaseCase := 0 TO 1 DO
			FOR operation := 0 TO 6 DO
				_CollisionDictionary.Clear();
				_CollisionSet.Clear();

				IF foundCase = 1 THEN
					_CollisionDictionary.SetCopy(key := _Scalar, value := _OtherScalar);
					_CollisionSet.SetCopy(value := _Scalar);
				END_IF

				_CloneExitCount := TOF_Core.UnsignedInt32.ZERO;

				IF ownedCase = 1 THEN
					prepareOwnedValue();
					_Query := _OwnedValue;
					_OwnedValue.Reset();
				ELSE
					_Query := TOF_Core.GenericValueFactory.FromParts(
						genericTypeClass := TOF_Core.GENERIC_TYPE_CLASS.OBJECT,
						address := _CloneSource.SelfAddress,
						size := _CloneSource.SelfSize,
						memoryManagementBehavior :=
							TOF_Core.GENERIC_MEMORY_MANAGEMENT_BEHAVIOR.STORE_ORIGINAL_REFERENCE_AND_NOT_OWNS_MEMORY
					);
				END_IF

				scenarioDescription := TOF_Core.WideStrings.Concat255(
					"Operation ",
					TO_WSTRING(operation),
					", found=",
					TO_WSTRING(foundCase),
					", owned=",
					TO_WSTRING(ownedCase),
					", release=",
					TO_WSTRING(releaseCase)
				);

				releaseQuery := releaseCase = 1;
				queryForCall := _Query;

				IF releaseQuery THEN
					// The receiving call is responsible for disposal even when its lookup fails.
					_Query.Reset();
				END_IF

				CASE operation OF
					0:
						found := _CollisionDictionary.ContainsGenericKey(key := queryForCall, releaseKey := releaseQuery);
					1:
						position := _CollisionDictionary.GetGenericKeyPosition(key := queryForCall, releaseKey := releaseQuery);
						found := position >= TOF_Core.SignedInt32.ZERO;
					2:
						found := _CollisionDictionary.TryGetValueByGenericKey(
							key := queryForCall,
							releaseKey := releaseQuery,
							value => foundValue
						);
					3:
						_CollisionDictionary.TryRemoveByGenericKey(
							key := queryForCall,
							releaseKey := releaseQuery,
							removed => found
						);
					4:
						found := _CollisionSet.ContainsGeneric(value := queryForCall, releaseValue := releaseQuery);
					5:
						position := _CollisionSet.GetGenericValuePosition(value := queryForCall, releaseValue := releaseQuery);
						found := position >= TOF_Core.SignedInt32.ZERO;
					6:
						_CollisionSet.TryRemoveGeneric(value := queryForCall, releaseValue := releaseQuery, removed => found);
				END_CASE

				queryForCall.Reset();

				_Assertions.ThatBool(
					actual := found,
					message := TOF_Core.WideStrings.Concat255(
						scenarioDescription,
						": ",
						"Owned and borrowed queries must preserve found and missing outcomes"
					)
				).ToBe(expected := foundCase = 1);
				_Assertions.ThatUDInt(
					actual := _CloneExitCount,
					message := TOF_Core.WideStrings.Concat255(
						scenarioDescription,
						": ",
						"Only an explicitly released owned query may be destroyed by lookup"
					)
				).ToBe(expected := TO_UDINT(ownedCase * releaseCase));

				IF NOT releaseQuery THEN
					IF ownedCase = 1 AND_THEN _CloneExitCount <> TOF_Core.UnsignedInt32.ZERO THEN
						// The count assertion above already reports unexpected destruction.
						_Query.Reset();
					ELSE
						_Assertions.ThatBool(
							actual := _Query.IsNull,
							message := TOF_Core.WideStrings.Concat255(
								scenarioDescription,
								": ",
								"Retained query descriptor must remain valid"
							)
						).IsFalse();
						queryAsInterface := _Query.AsIObject();
						_Assertions.ThatBool(
							actual := queryAsInterface <> 0,
							message := TOF_Core.WideStrings.Concat255(
								scenarioDescription,
								": ",
								"Retained query object must remain alive"
							)
						).IsTrue();
						_Query.Release();
					END_IF
				END_IF

				_Assertions.ThatUDInt(
					actual := _CloneExitCount,
					message := TOF_Core.WideStrings.Concat255(
						scenarioDescription,
						": ",
						"Each owned query must have exactly one disposal owner"
					)
				).ToBe(expected := TO_UDINT(ownedCase));
			END_FOR
		END_FOR
	END_FOR
END_FOR
END_METHOD

(*!
<summary>Preserves collision chains through growth, middle removal, reinsertion and reuse.</summary>
<description>
Starts with independent fixture state. The harness clears persistent resources before publication, including
after an aborted call. Terminal OOM injection is reserved for an isolated test.
</description>
*)
METHOD PRIVATE hashCollisionGrowth
VAR
	i : DINT;
	removed : BOOL;
	foundValue : TOF_Core.GENERIC_VALUE;
END_VAR
_CollisionDictionary.DefaultDynamicAllocationElementCount := 2;
_CollisionSet.DefaultDynamicAllocationElementCount := 2;

FOR i := 1 TO 25 DO
	_CollisionDictionary.SetCopy(key := i, value := i);
	_CollisionSet.SetCopy(value := i);
END_FOR

_Assertions.ThatDInt(
	actual := _CollisionDictionary.Length,
	message := "All dictionary collisions must fit"
).ToBe(expected := 25);
_Assertions.ThatDInt(
	actual := _CollisionSet.Length,
	message := "All set collisions must fit"
).ToBe(expected := 25);

FOR i := 1 TO 25 DO
	_Assertions.ThatBool(
		actual := _CollisionDictionary.TryGetValueByKey(key := i, value => foundValue),
		message := "Growth must retain each dictionary collision"
	).IsTrue();
	_Assertions.ThatDInt(
		actual := foundValue.AsDInt(),
		message := "Dictionary collision value must match"
	).ToBe(expected := i);
	_Assertions.ThatBool(
		actual := _CollisionSet.Contains(value := i),
		message := "Growth must retain each set collision"
	).IsTrue();
END_FOR

_CollisionDictionary.TryRemoveByKey(key := _MiddleScalar, removed => removed);
_Assertions.ThatBool(
	actual := removed,
	message := "Middle collision must be removed"
).IsTrue();
_CollisionSet.TryRemove(value := _MiddleScalar, removed => removed);
_Assertions.ThatBool(
	actual := removed,
	message := "Middle set collision must be removed"
).IsTrue();
_Assertions.ThatBool(
	actual := _CollisionDictionary.ContainsKey(key := _MiddleScalar),
	message := "Removed key must be absent"
).IsFalse();
_Assertions.ThatBool(
	actual := _CollisionSet.Contains(value := _MiddleScalar),
	message := "Removed value must be absent"
).IsFalse();
_CollisionDictionary.SetCopy(key := _MiddleScalar, value := _OtherScalar);
_CollisionSet.SetCopy(value := _MiddleScalar);

